# B&R Automation Studio project reAM250plc (part 3)

#### IOModule_X20AT6402.hpp
```cpp
/*++

Copyright (C) 2024 Institute for Machine Tools and Industrial Management
TUM School of Engineering and Design
Technical University of Munich

All rights reserved.

Redistribution and use in source and binary forms, with or without
modification, are permitted provided that the following conditions are met:
	* Redistributions of source code must retain the above copyright
	  notice, this list of conditions and the following disclaimer.
	* Redistributions in binary form must reproduce the above copyright
	  notice, this list of conditions and the following disclaimer in the
	  documentation and/or other materials provided with the distribution.
	* Neither the name of the Technical University of Munich nor the
	  names of its contributors may be used to endorse or promote products
	  derived from this software without specific prior written permission.

THIS SOFTWARE IS PROVIDED BY THE COPYRIGHT HOLDERS AND CONTRIBUTORS "AS IS" AND
ANY EXPRESS OR IMPLIED WARRANTIES, INCLUDING, BUT NOT LIMITED TO, THE IMPLIED
WARRANTIES OF MERCHANTABILITY AND FITNESS FOR A PARTICULAR PURPOSE ARE
DISCLAIMED. IN NO EVENT SHALL TECHNICAL UNIVERSITY OF MUNICH BE LIABLE FOR ANY
DIRECT, INDIRECT, INCIDENTAL, SPECIAL, EXEMPLARY, OR CONSEQUENTIAL DAMAGES
(INCLUDING, BUT NOT LIMITED TO, PROCUREMENT OF SUBSTITUTE GOODS OR SERVICES;
LOSS OF USE, DATA, OR PROFITS; OR BUSINESS INTERRUPTION) HOWEVER CAUSED AND
ON ANY THEORY OF LIABILITY, WHETHER IN CONTRACT, STRICT LIABILITY, OR TORT
(INCLUDING NEGLIGENCE OR OTHERWISE) ARISING IN ANY WAY OUT OF THE USE OF THIS
SOFTWARE, EVEN IF ADVISED OF THE POSSIBILITY OF SUCH DAMAGE.

*/

#ifndef __IOMODULE_X20AT6402_HPP
#define __IOMODULE_X20AT6402_HPP

#include "../Framework/Framework.hpp"

namespace BuRCPP {

	enum class eIOModuleType_X20AT6402 : uint32_t {
		mtUnknown = 0,
		mtVoltage10V = 1,
		mtCurrent20mA = 2,
		mtCurrent24mA = 3
	};

	class CIOModule_X20AT6402 : public CIOModule {
		protected:
		IOMappingX20AT6402_TYP * m_pMapping;
		eIOModuleType_X20AT6402 m_ModuleType;
		int16_t m_nLowerLimit;
		int16_t m_nUpperLimit;

		public:
		CIOModule_X20AT6402 (const std::string & sName, IOMappingX20AT6402_TYP * pMapping);
		virtual ~CIOModule_X20AT6402 ();

		bool isActive () override;
		uint32_t getSerialNumber () override;
		uint16_t getModuleID () override;
		uint16_t getHardwareVariant () override;
		uint16_t getFirmwareVersion () override;

		int16_t getRawValue (uint32_t nChannelNo);
		;
		uint16_t getIOStatus (uint32_t nChannelNo);

		virtual void onRegisterJournal () override;
		virtual void onUpdateJournal () override;

	};

}

#endif //__IOMODULE_X20AT6402_HPP
```

#### IOModule_X20AT6402.cpp
```cpp
/*++

Copyright (C) 2024 Institute for Machine Tools and Industrial Management
TUM School of Engineering and Design
Technical University of Munich

All rights reserved.

Redistribution and use in source and binary forms, with or without
modification, are permitted provided that the following conditions are met:
	* Redistributions of source code must retain the above copyright
	  notice, this list of conditions and the following disclaimer.
	* Redistributions in binary form must reproduce the above copyright
	  notice, this list of conditions and the following disclaimer in the
	  documentation and/or other materials provided with the distribution.
	* Neither the name of the Technical University of Munich nor the
	  names of its contributors may be used to endorse or promote products
	  derived from this software without specific prior written permission.

THIS SOFTWARE IS PROVIDED BY THE COPYRIGHT HOLDERS AND CONTRIBUTORS "AS IS" AND
ANY EXPRESS OR IMPLIED WARRANTIES, INCLUDING, BUT NOT LIMITED TO, THE IMPLIED
WARRANTIES OF MERCHANTABILITY AND FITNESS FOR A PARTICULAR PURPOSE ARE
DISCLAIMED. IN NO EVENT SHALL TECHNICAL UNIVERSITY OF MUNICH BE LIABLE FOR ANY
DIRECT, INDIRECT, INCIDENTAL, SPECIAL, EXEMPLARY, OR CONSEQUENTIAL DAMAGES
(INCLUDING, BUT NOT LIMITED TO, PROCUREMENT OF SUBSTITUTE GOODS OR SERVICES;
LOSS OF USE, DATA, OR PROFITS; OR BUSINESS INTERRUPTION) HOWEVER CAUSED AND
ON ANY THEORY OF LIABILITY, WHETHER IN CONTRACT, STRICT LIABILITY, OR TORT
(INCLUDING NEGLIGENCE OR OTHERWISE) ARISING IN ANY WAY OUT OF THE USE OF THIS
SOFTWARE, EVEN IF ADVISED OF THE POSSIBILITY OF SUCH DAMAGE.

*/

#include "IOModule_X20AT6402.hpp"

// Raw Registers
#define JOURNALVARIABLE_X20AT6402_MODULEOK 1
#define JOURNALVARIABLE_X20AT6402_SERIALNUMBER 2
#define JOURNALVARIABLE_X20AT6402_MODULEID 3
#define JOURNALVARIABLE_X20AT6402_HARDWAREVARIANT 4
#define JOURNALVARIABLE_X20AT6402_FIRMWAREVERSION 5
#define JOURNALVARIABLE_X20AT6402_TEMPERATURE01 6
#define JOURNALVARIABLE_X20AT6402_TEMPERATURE02 7
#define JOURNALVARIABLE_X20AT6402_TEMPERATURE03 8
#define JOURNALVARIABLE_X20AT6402_TEMPERATURE04 9
#define JOURNALVARIABLE_X20AT6402_TEMPERATURE05 10
#define JOURNALVARIABLE_X20AT6402_TEMPERATURE06 11
#define JOURNALVARIABLE_X20AT6402_STATUSINPUT01 12
#define JOURNALVARIABLE_X20AT6402_STATUSINPUT02 13

namespace BuRCPP {

	CIOModule_X20AT6402	::CIOModule_X20AT6402 (const std::string & sName, IOMappingX20AT6402_TYP * pMapping)
		: CIOModule (sName), m_pMapping (pMapping)
	{

	}

	CIOModule_X20AT6402::~CIOModule_X20AT6402 ()
	{
	}

	void CIOModule_X20AT6402::onRegisterJournal ()
	{
		registerBoolValue ("ModuleOk", JOURNALVARIABLE_X20AT6402_MODULEOK);
		registerUInt32Value ("SerialNumber", JOURNALVARIABLE_X20AT6402_SERIALNUMBER);
		registerUInt16Value ("ModuleID", JOURNALVARIABLE_X20AT6402_MODULEID);
		registerUInt16Value ("HardwareVariant", JOURNALVARIABLE_X20AT6402_HARDWAREVARIANT);
		registerUInt16Value ("FirmwareVersion", JOURNALVARIABLE_X20AT6402_FIRMWAREVERSION);
		registerInt16Value ("Temperature01", JOURNALVARIABLE_X20AT6402_TEMPERATURE01);
		registerInt16Value ("Temperature02", JOURNALVARIABLE_X20AT6402_TEMPERATURE02);
		registerInt16Value ("Temperature03", JOURNALVARIABLE_X20AT6402_TEMPERATURE03);
		registerInt16Value ("Temperature04", JOURNALVARIABLE_X20AT6402_TEMPERATURE04);
		registerInt16Value ("Temperature05", JOURNALVARIABLE_X20AT6402_TEMPERATURE05);
		registerInt16Value ("Temperature06", JOURNALVARIABLE_X20AT6402_TEMPERATURE06);
		registerUInt8Value ("StatusInput01", JOURNALVARIABLE_X20AT6402_STATUSINPUT01);
		registerUInt8Value ("StatusInput02", JOURNALVARIABLE_X20AT6402_STATUSINPUT02);
	}

	void CIOModule_X20AT6402::onUpdateJournal ()
	{
		setBoolValue (JOURNALVARIABLE_X20AT6402_MODULEOK, m_pMapping->ModuleOk);
		setIntegerValue (JOURNALVARIABLE_X20AT6402_SERIALNUMBER, m_pMapping->SerialNumber);
		setIntegerValue (JOURNALVARIABLE_X20AT6402_MODULEID, m_pMapping->ModuleID);
		setIntegerValue (JOURNALVARIABLE_X20AT6402_HARDWAREVARIANT, m_pMapping->HardwareVariant);
		setIntegerValue (JOURNALVARIABLE_X20AT6402_FIRMWAREVERSION, m_pMapping->FirmwareVersion);
		setIntegerValue (JOURNALVARIABLE_X20AT6402_TEMPERATURE01, m_pMapping->Temperature01);
		setIntegerValue (JOURNALVARIABLE_X20AT6402_TEMPERATURE02, m_pMapping->Temperature02);
		setIntegerValue (JOURNALVARIABLE_X20AT6402_TEMPERATURE03, m_pMapping->Temperature03);
		setIntegerValue (JOURNALVARIABLE_X20AT6402_TEMPERATURE04, m_pMapping->Temperature04);
		setIntegerValue (JOURNALVARIABLE_X20AT6402_TEMPERATURE05, m_pMapping->Temperature05);
		setIntegerValue (JOURNALVARIABLE_X20AT6402_TEMPERATURE06, m_pMapping->Temperature06);
		setIntegerValue (JOURNALVARIABLE_X20AT6402_STATUSINPUT01, m_pMapping->StatusInput01);
		setIntegerValue (JOURNALVARIABLE_X20AT6402_STATUSINPUT02, m_pMapping->StatusInput02);
	}

	bool CIOModule_X20AT6402::isActive ()
	{
		return m_pMapping->ModuleOk != 0;
	}

	uint32_t CIOModule_X20AT6402::getSerialNumber ()
	{
		return m_pMapping->SerialNumber;
	}

	uint16_t CIOModule_X20AT6402::getModuleID ()
	{
		return m_pMapping->ModuleID;
	}

	uint16_t CIOModule_X20AT6402::getHardwareVariant ()
	{
		return m_pMapping->HardwareVariant;
	}

	uint16_t CIOModule_X20AT6402::getFirmwareVersion ()
	{
		return m_pMapping->FirmwareVersion;
	}

	int16_t CIOModule_X20AT6402::getRawValue (uint32_t nChannelNo)
	{

		switch (nChannelNo) {
			case 1: return m_pMapping->Temperature01;
			case 2: return m_pMapping->Temperature02;
			case 3: return m_pMapping->Temperature03;
			case 4: return m_pMapping->Temperature04;
			case 5: return m_pMapping->Temperature05;
			case 6: return m_pMapping->Temperature06;
			default:
				throw CException (eErrorCode::INVALIDCHANNELNUMBER, "invalid channel number: " + std::to_string (nChannelNo));
		}
	}

	uint16_t CIOModule_X20AT6402::getIOStatus (uint32_t nChannelNo)
	{
		//status IDs: 0 = no error, 1 = lower limit value undershot, 2 = upper limit value exceeded, 3 = wire breakage
		switch (nChannelNo) {
			case 1: return (m_pMapping->StatusInput01 & 0x03);
			case 2: return ((m_pMapping->StatusInput01 >> 2) & 0x03);
			case 3: return ((m_pMapping->StatusInput01 >> 4) & 0x03);
			case 4: return ((m_pMapping->StatusInput01 >> 6) & 0x03);
			case 5: return (m_pMapping->StatusInput02 & 0x03);
			case 6: return ((m_pMapping->StatusInput02 >> 2) & 0x03);
			default:
				throw CException (eErrorCode::INVALIDCHANNELNUMBER, "invalid channel number: " + std::to_string (nChannelNo));
		}
	}

}
```

#### MappMotion_SingleAxis.hpp
```cpp
/*++

Copyright (C) 2024 Institute for Machine Tools and Industrial Management
TUM School of Engineering and Design
Technical University of Munich

All rights reserved.

Redistribution and use in source and binary forms, with or without
modification, are permitted provided that the following conditions are met:
	* Redistributions of source code must retain the above copyright
	  notice, this list of conditions and the following disclaimer.
	* Redistributions in binary form must reproduce the above copyright
	  notice, this list of conditions and the following disclaimer in the
	  documentation and/or other materials provided with the distribution.
	* Neither the name of the Technical University of Munich nor the
	  names of its contributors may be used to endorse or promote products
	  derived from this software without specific prior written permission.

THIS SOFTWARE IS PROVIDED BY THE COPYRIGHT HOLDERS AND CONTRIBUTORS "AS IS" AND
ANY EXPRESS OR IMPLIED WARRANTIES, INCLUDING, BUT NOT LIMITED TO, THE IMPLIED
WARRANTIES OF MERCHANTABILITY AND FITNESS FOR A PARTICULAR PURPOSE ARE
DISCLAIMED. IN NO EVENT SHALL TECHNICAL UNIVERSITY OF MUNICH BE LIABLE FOR ANY
DIRECT, INDIRECT, INCIDENTAL, SPECIAL, EXEMPLARY, OR CONSEQUENTIAL DAMAGES
(INCLUDING, BUT NOT LIMITED TO, PROCUREMENT OF SUBSTITUTE GOODS OR SERVICES;
LOSS OF USE, DATA, OR PROFITS; OR BUSINESS INTERRUPTION) HOWEVER CAUSED AND
ON ANY THEORY OF LIABILITY, WHETHER IN CONTRACT, STRICT LIABILITY, OR TORT
(INCLUDING NEGLIGENCE OR OTHERWISE) ARISING IN ANY WAY OUT OF THE USE OF THIS
SOFTWARE, EVEN IF ADVISED OF THE POSSIBILITY OF SUCH DAMAGE.

*/

#ifndef __MAPPMOTION_SINGLEAXIS_HPP
#define __MAPPMOTION_SINGLEAXIS_HPP

#include "../Framework/Framework.hpp"
#include <memory>

namespace BuRCPP {

	class CMappMotion_SingleAxisImpl;

	enum class eMappMotion_SingleAxisType : int32_t {
		mtLinearAxis = 0,
		mtRotationalAxis = 1,
	};

//	enum class eMappMotion_SingleLinearAxisHomingMode : int32_t {
//		mtDefault = 0,
//		mtRestorePosition = 1,
//	};

	enum class eMappMotion_SingleAxisState : int32_t {
		UNKNOWN = 0,
		STATE_IDLE = 1,
		STATE_SETTINGPOWERON = 2,
		STATE_SETTINGPOWEROFF = 3,
		STATE_REFERENCING = 4,
		STATE_INITABSOLUTEMOVEMENT = 5,
		STATE_INITRELATIVEMOVEMENT = 6,
		STATE_INITVELOCITYMOVEMENT = 7,
		STATE_WAITINGFORMOVEMENT = 8,
		STATE_SETTINGPOWERON_TO_REFERENCE = 9,
		STATE_ERROR = 255,
	};

	class CMappMotion_SingleAxis : public CAxisModule {
		protected:
		McHomingModeEnum m_HomingMode;

		std::shared_ptr<CMappMotion_SingleAxisImpl> m_pImpl;
		eMappMotion_SingleAxisType m_Type;
		eMappMotion_SingleAxisState m_State;

		double m_dSpeedInMMperSecondToSet;
		double m_dAccelerationInMMPerSecondSquaredToSet;
		double m_dTargetPositionInMMToSet;
		double m_dDistanceInMMToSet;

		double m_dSpeedInDegreeperSecondToSet;
		double m_dAccelerationInDegreePerSecondSquaredToSet;
		double m_dTargetPositionInDegreeToSet;
		double m_dDistanceInDegreeToSet;

		public:

		CMappMotion_SingleAxis (const std::string & sName, void * pLink);
		virtual ~CMappMotion_SingleAxis ();

		bool isActive () override;
		bool isIdle ();

		virtual ePLCOpenAxisState getPLCOpenState () override;
		virtual bool isPowered () override;
		virtual bool isReferenced () override;
		virtual bool isMoving () override;
	//	virtual bool isMoveDone () override;

		virtual bool canSetPower () override;
		virtual void setPower (bool bPowerOn) override;

		virtual bool canReference () override;
		virtual void startReference () override;

		virtual void setPowerOnAndStartReference () override;

		void setHomingMode (McHomingModeEnum homingMode);

		virtual bool canMoveAxis ();

		void resetError ();
		void moveAxisReset ();
		bool isError ();
		bool isInPosition ();

		virtual void handleCyclic () override;

		virtual void * getFunctionBlockPtr ();

		virtual void * getParameterBlockPtr ();

		virtual void onRegisterJournal () override;
		virtual void onUpdateJournal () override;

	};

	class CMappMotion_SingleRotationalAxis : public CMappMotion_SingleAxis
	{
		private:

		double m_dMinSpeedInDegreeperSecond;
		double m_dMaxSpeedInDegreeperSecond;

		double m_dMinAccelerationInDegreeperSecond;
		double m_dMaxAccelerationInDegreeperSecond;

		public:

		CMappMotion_SingleRotationalAxis (const std::string & sName, void * pLink);
		virtual ~CMappMotion_SingleRotationalAxis ();

		void moveAxisAbsolute (double targetPositionInDegree, double speedInDegreeperSecond, double accelerationinDegreeSecondsSquared);
		void moveAxisRelative (double targetPositionInDegree, double speedInDegreeperSecond, double accelerationinDegreeSecondsSquared);
		void moveAxisVelocity (double speedInDegreeperSecond, double accelerationinDegreeSecondsSquared);

		double getCurrentPositionInDegree ();
		double getCurrentVelocityInDegreePerSecond ();
	};
	class CMappMotion_SingleLinearAxis : public CMappMotion_SingleAxis
	{
		private:

		double m_dMinSpeedInMMperSecond;
		double m_dMaxSpeedInMMperSecond;

		double m_dMinAccelerationInMMperSecond;
		double m_dMaxAccelerationInMMperSecond;

		public:

		CMappMotion_SingleLinearAxis (const std::string & sName, void * pLink);
		virtual ~CMappMotion_SingleLinearAxis ();

		void moveAxisAbsolute (double targetPositionInMM, double speedInMMperSecond, double accelerationInMMPerSecondSquared);
		void moveAxisRelative (double targetPositionInMM, double speedInMMperSecond, double accelerationInMMPerSecondSquared);
		void moveAxisVelocity (double speedInMMperSecond, double accelerationInMMPerSecondSquared);

		double getCurrentPositionInMM ();
		double getCurrentVelocityInMMPerSecond ();

	};

}

#endif // __MAPPMOTION_SINGLEAXIS_HPP
```

#### MappMotion_SingleAxis.cpp
```cpp
/*++

Copyright (C) 2024 Institute for Machine Tools and Industrial Management
TUM School of Engineering and Design
Technical University of Munich

All rights reserved.

Redistribution and use in source and binary forms, with or without
modification, are permitted provided that the following conditions are met:
	* Redistributions of source code must retain the above copyright
	  notice, this list of conditions and the following disclaimer.
	* Redistributions in binary form must reproduce the above copyright
	  notice, this list of conditions and the following disclaimer in the
	  documentation and/or other materials provided with the distribution.
	* Neither the name of the Technical University of Munich nor the
	  names of its contributors may be used to endorse or promote products
	  derived from this software without specific prior written permission.

THIS SOFTWARE IS PROVIDED BY THE COPYRIGHT HOLDERS AND CONTRIBUTORS "AS IS" AND
ANY EXPRESS OR IMPLIED WARRANTIES, INCLUDING, BUT NOT LIMITED TO, THE IMPLIED
WARRANTIES OF MERCHANTABILITY AND FITNESS FOR A PARTICULAR PURPOSE ARE
DISCLAIMED. IN NO EVENT SHALL TECHNICAL UNIVERSITY OF MUNICH BE LIABLE FOR ANY
DIRECT, INDIRECT, INCIDENTAL, SPECIAL, EXEMPLARY, OR CONSEQUENTIAL DAMAGES
(INCLUDING, BUT NOT LIMITED TO, PROCUREMENT OF SUBSTITUTE GOODS OR SERVICES;
LOSS OF USE, DATA, OR PROFITS; OR BUSINESS INTERRUPTION) HOWEVER CAUSED AND
ON ANY THEORY OF LIABILITY, WHETHER IN CONTRACT, STRICT LIABILITY, OR TORT
(INCLUDING NEGLIGENCE OR OTHERWISE) ARISING IN ANY WAY OUT OF THE USE OF THIS
SOFTWARE, EVEN IF ADVISED OF THE POSSIBILITY OF SUCH DAMAGE.

*/
#include "MappMotion_SingleAxis.hpp"

#include <bur/plctypes.h>

#ifdef _DEFAULT_INCLUDES
#include <AsDefault.h>
#endif

#include <string.h>

#define MAPPMOTION_LINEARAXIS_DEFAULTMINSPEED_IN_MMPERSECOND 0.001f
#define MAPPMOTION_LINEARAXIS_DEFAULTMAXSPEED_IN_MMPERSECOND 1000000.0f
#define MAPPMOTION_LINEARAXIS_DEFAULTMINACCELERATION_IN_MMPERSECONDSQUARED 0.001f
#define MAPPMOTION_LINEARAXIS_DEFAULTMAXACCELERATION_IN_MMPERSECONDSQUARED 1000000.0f

#define MAPPMOTION_ROTARYAXIS_DEFAULTMINSPEED_IN_DEGREEPERSECOND 0.001f
#define MAPPMOTION_ROTARYAXIS_DEFAULTMAXSPEED_IN_DEGREEPERSECOND 1000000.0f
#define MAPPMOTION_ROTARYAXIS_DEFAULTMINACCELERATION_IN_DEGREEPERSECONDSQUARED 0.001f
#define MAPPMOTION_ROTARYAXIS_DEFAULTMAXACCELERATION_IN_DEGREEPERSECONDSQUARED 1000000.0f

#define JOURNALVARIABLE_AXIS_PLCOPENSTATE 1
#define JOURNALVARIABLE_AXIS_CANSETPOWER 2
#define JOURNALVARIABLE_AXIS_ISPOWERED 3
#define JOURNALVARIABLE_AXIS_ISREFERENCED 4
#define JOURNALVARIABLE_AXIS_ISMOVING 5
#define JOURNALVARIABLE_AXIS_ISINPOSITION 6
#define JOURNALVARIABLE_AXIS_ACTUALPOSITION 7
#define JOURNALVARIABLE_AXIS_ACTUALVELOCITY 8

namespace BuRCPP {

	class CMappMotion_SingleAxisImpl {
		private:
		MpAxisBasicParType m_Parameters;
		MpAxisBasic_typ m_FunctionBlock;
		public:

		CMappMotion_SingleAxisImpl (McAxisType * pLink)
		{
			memset ((void*) &m_Parameters, 0, sizeof (MpAxisBasicParType));
			memset ((void*) &m_FunctionBlock, 0, sizeof (MpAxisBasic_typ));

			m_FunctionBlock.MpLink = pLink;
			m_FunctionBlock.Parameters = &m_Parameters;
			m_FunctionBlock.Enable = true;
		}

		virtual ~CMappMotion_SingleAxisImpl ()
		{
			memset ((void*) &m_Parameters, 0, sizeof (MpAxisBasicParType));
			memset ((void*) &m_FunctionBlock, 0, sizeof (MpAxisBasic_typ));
		}

		int32_t getPLCOpenState () const
		{
			return m_FunctionBlock.Info.PLCopenState;
		}

		bool isError () const
		{
			return m_FunctionBlock.Error;
		}

		bool canSetPower () const
		{
			return m_FunctionBlock.Info.ReadyToPowerOn;
		}

		bool isPowered () const
		{
			return m_FunctionBlock.PowerOn;
		}

		bool isReferenced () const
		{
			return m_FunctionBlock.IsHomed;
		}

		bool isMoving () const
		{
			return m_FunctionBlock.MoveActive;
		}

		bool isInPosition () const
		{
			return m_FunctionBlock.InPosition;
		}

		float getCurrentPosition () const
		{
			return m_FunctionBlock.Position;
		}

		float getCurrentVelocity () const
		{
			return m_FunctionBlock.Velocity;
		}

		void setErrorResetFlag (bool bErrorResetFlag)
		{
			m_FunctionBlock.ErrorReset = bErrorResetFlag;
		}

		void setPowerFlag (bool bPowerFlag)
		{
			m_FunctionBlock.Power = bPowerFlag;
		}

		void setHomeFlag (bool bHomeFlag)
		{
			m_FunctionBlock.Home = bHomeFlag;
		}

		void setVelocityParameter (float fVelocity)
		{
			m_Parameters.Velocity = fVelocity;
		}

		void setAccelerationDecelerationParameter (float fAccelerationDeceleration)
		{
			m_Parameters.Acceleration = fAccelerationDeceleration;
			m_Parameters.Deceleration = fAccelerationDeceleration;
		}

		void setAbsoluteMovementTarget (float fTargetPosition)
		{
			m_Parameters.Position = fTargetPosition;
		}

		void setAbsoluteMovementFlag (bool bMovementFlag)
		{
			m_FunctionBlock.MoveAbsolute = bMovementFlag;
		}

		void setRelativeMovementDistance (float fRelativeDistance)
		{
			m_Parameters.Distance = fRelativeDistance;
		}

		void setRelativeMovementFlag (bool bMovementFlag)
		{
			m_FunctionBlock.MoveAdditive = bMovementFlag;
		}

		void setVelocityMovementFlag (bool bMovementFlag)
		{
			m_FunctionBlock.MoveVelocity = bMovementFlag;
		}

		void setHomingMode (McHomingModeEnum homingMode)
		{
			m_Parameters.Homing.Mode = homingMode;
		}

		void handleCyclic ()
		{
			MpAxisBasic(&m_FunctionBlock);
		}

		void * getFunctionBlockPtr ()
		{
			return &m_FunctionBlock;
		}

		void * getParameterBlockPtr ()
		{
			return &m_Parameters;
		}

	};

	CMappMotion_SingleAxis::CMappMotion_SingleAxis (const std::string & sName, void * pLink)
		: CAxisModule (sName),
		m_State (eMappMotion_SingleAxisState::STATE_IDLE),
		m_dSpeedInMMperSecondToSet (0.0),
		m_dAccelerationInMMPerSecondSquaredToSet (0.0),
		m_dTargetPositionInMMToSet (0.0),
		m_dDistanceInMMToSet (0.0)
	{
		m_HomingMode = mcHOMING_DEFAULT;

		if (pLink == nullptr)
			throw CException (eErrorCode::INVALIDAXISLINK, "invalid axis link: " + sName);
/*	if (pFunctionBlock == nullptr)
		throw CException (eErrorCode::INVALIDFUNCTIONBLOCK, "invalid axis function block: " + sName);
	if (pParameterBlock == nullptr)
		throw CException (eErrorCode::INVALIDPARAMETERBLOCK, "invalid axis parameter block: " + sName);*/

		m_pImpl.reset ( new CMappMotion_SingleAxisImpl ((McAxisType*) pLink) );

		// TODO: Read out speed and acceleration limits...
	}

	CMappMotion_SingleAxis::~CMappMotion_SingleAxis ()
	{
	}

	void * CMappMotion_SingleAxis::getFunctionBlockPtr ()
	{
		return m_pImpl->getFunctionBlockPtr ();
	}

	void * CMappMotion_SingleAxis::getParameterBlockPtr ()
	{
		return m_pImpl->getParameterBlockPtr ();
	}

	bool CMappMotion_SingleAxis::isActive ()
	{
		return true;
	}

	ePLCOpenAxisState CMappMotion_SingleAxis::getPLCOpenState ()
	{
		return (ePLCOpenAxisState) m_pImpl->getPLCOpenState ();

	}

	bool CMappMotion_SingleAxis::isIdle ()
	{
		return (m_State == eMappMotion_SingleAxisState::STATE_IDLE);
	}

	bool CMappMotion_SingleAxis::isPowered ()
	{
		return m_pImpl->isPowered ();
	}

	bool CMappMotion_SingleAxis::isReferenced ()
	{
		return m_pImpl->isReferenced ();
	}

	bool CMappMotion_SingleAxis::isMoving ()
	{
		return m_pImpl->isMoving ();
	}

	bool CMappMotion_SingleAxis::isInPosition ()
	{
		return m_pImpl->isInPosition ();
	}

	bool CMappMotion_SingleAxis::canSetPower ()
	{
		return m_pImpl->canSetPower ();
	}

	bool CMappMotion_SingleAxis::isError ()
	{
		return m_pImpl->isError ();
	}

	void CMappMotion_SingleAxis::setPower (bool bPowerOn)
	{
		if (bPowerOn) {
			if (canSetPower ()) {
				m_pImpl->setPowerFlag (true);
				m_State = eMappMotion_SingleAxisState::STATE_SETTINGPOWERON;
			} else {
				throw CException (eErrorCode::COULDNOTPOWERAXIS, "could not power axis: " + m_sName);
			}

		}
		else {
			if (isIdle ()) {
				m_pImpl->setPowerFlag (false);
				m_State = eMappMotion_SingleAxisState::STATE_SETTINGPOWEROFF;

			} else {
				throw CException (eErrorCode::COULDNOTPOWERAXIS, "could not gracefully unpower axis: " + m_sName);
			}
		}

	}

	bool CMappMotion_SingleAxis::canReference ()
	{
		if (isIdle () && isPowered () && (m_pImpl->getPLCOpenState () == mcAXIS_STANDSTILL)) {
			return true;
		} else {
			return false;
		}
	}

	void CMappMotion_SingleAxis::startReference ()
	{
		if (canReference ()) {

			if (DiagCpuIsSimulated()) {
				m_HomingMode = mcHOMING_DIRECT;
				m_pImpl->setHomingMode(m_HomingMode);

			}
			else
			{
				m_pImpl->setHomingMode(m_HomingMode);
			}

			m_pImpl->setHomeFlag (true);
			m_State = eMappMotion_SingleAxisState::STATE_REFERENCING;

		} else {

			throw CException (eErrorCode::COULDNOTREFERENCEAXIS, "could not reference axis: " + m_sName);

		}
	}

	void CMappMotion_SingleAxis::setHomingMode (McHomingModeEnum homingMode)
	{
		m_HomingMode = homingMode;
		m_pImpl->setHomingMode(m_HomingMode);
	}

	void CMappMotion_SingleAxis::setPowerOnAndStartReference ()
	{
		if (canSetPower ()) {
			m_pImpl->setPowerFlag (true);
			m_State = eMappMotion_SingleAxisState::STATE_SETTINGPOWERON_TO_REFERENCE;
		} else {
			throw CException (eErrorCode::COULDNOTPOWERAXIS, "could not power axis: " + m_sName);
		}
	}

	bool CMappMotion_SingleAxis::canMoveAxis ()
	{
		if (isIdle () && isPowered () && isReferenced() && (m_pImpl->getPLCOpenState () == mcAXIS_STANDSTILL)) {
			return true;
		} else {
			return false;
		}
	}

	void CMappMotion_SingleAxis::resetError ()
	{
		if (m_pImpl->isError ()) {
			m_pImpl->setPowerFlag(false);
			m_pImpl->setErrorResetFlag (true);
		}
		else{
			m_pImpl->setErrorResetFlag (false);
			m_pImpl->setPowerFlag(true);
			m_State = eMappMotion_SingleAxisState::STATE_SETTINGPOWERON;
		}

	}

	void CMappMotion_SingleAxis::moveAxisReset ()
	{
		m_pImpl->setVelocityMovementFlag(false);
		m_pImpl->setAbsoluteMovementFlag(false);
		m_pImpl->setRelativeMovementFlag(false);
	}

	void CMappMotion_SingleAxis::onRegisterJournal ()
	{
		registerUInt16Value ("PlcOpenState", JOURNALVARIABLE_AXIS_PLCOPENSTATE);
		registerBoolValue ("CanSetPower", JOURNALVARIABLE_AXIS_CANSETPOWER);
		registerBoolValue ("IsPowered", JOURNALVARIABLE_AXIS_ISPOWERED);
		registerBoolValue ("IsReferenced", JOURNALVARIABLE_AXIS_ISREFERENCED);
		registerBoolValue ("IsMoving", JOURNALVARIABLE_AXIS_ISMOVING);
		registerBoolValue ("IsInPosition", JOURNALVARIABLE_AXIS_ISINPOSITION);
		registerDoubleValue ("ActualPosition", JOURNALVARIABLE_AXIS_ACTUALPOSITION, -1000000, 1000000, 1);
		registerDoubleValue ("ActualVelocity", JOURNALVARIABLE_AXIS_ACTUALVELOCITY, -1000000, 1000000, 1);

	}

void CMappMotion_SingleAxis::onUpdateJournal ()
	{
		setIntegerValue (JOURNALVARIABLE_AXIS_PLCOPENSTATE, m_pImpl->getPLCOpenState());
		setBoolValue (JOURNALVARIABLE_AXIS_CANSETPOWER, canSetPower());
		setBoolValue (JOURNALVARIABLE_AXIS_ISPOWERED, isPowered());
		setBoolValue (JOURNALVARIABLE_AXIS_ISREFERENCED, isReferenced());
		setBoolValue (JOURNALVARIABLE_AXIS_ISMOVING, isMoving());
		setBoolValue (JOURNALVARIABLE_AXIS_ISINPOSITION,  isInPosition());
		setDoubleValue (JOURNALVARIABLE_AXIS_ACTUALPOSITION, m_pImpl->getCurrentPosition());
		setDoubleValue (JOURNALVARIABLE_AXIS_ACTUALVELOCITY, m_pImpl->getCurrentVelocity());

	}

CMappMotion_SingleLinearAxis::CMappMotion_SingleLinearAxis (const std::string & sName, void * pLink)
	: CMappMotion_SingleAxis (sName, pLink),
	m_dMinSpeedInMMperSecond (MAPPMOTION_LINEARAXIS_DEFAULTMINSPEED_IN_MMPERSECOND),
	m_dMaxSpeedInMMperSecond (MAPPMOTION_LINEARAXIS_DEFAULTMAXSPEED_IN_MMPERSECOND),
	m_dMinAccelerationInMMperSecond (MAPPMOTION_LINEARAXIS_DEFAULTMINACCELERATION_IN_MMPERSECONDSQUARED),
	m_dMaxAccelerationInMMperSecond (MAPPMOTION_LINEARAXIS_DEFAULTMAXACCELERATION_IN_MMPERSECONDSQUARED)
{
		m_Type = eMappMotion_SingleAxisType::mtLinearAxis;
}

CMappMotion_SingleLinearAxis::~CMappMotion_SingleLinearAxis ()
{
}

void CMappMotion_SingleLinearAxis::moveAxisAbsolute (double targetPositionInMM, double speedInMMperSecond, double accelerationInMMPerSecondSquared)
{
	if ((speedInMMperSecond < m_dMinSpeedInMMperSecond) || (speedInMMperSecond > m_dMaxSpeedInMMperSecond))
		throw CException (eErrorCode::INVALIDSPEEDVALUE, "invalid speed value for axis: " + m_sName);
	if ((accelerationInMMPerSecondSquared < m_dMinAccelerationInMMperSecond) || (accelerationInMMPerSecondSquared > m_dMaxAccelerationInMMperSecond))
		throw CException (eErrorCode::INVALIDACCELERATIONVALUE, "invalid acceleration value for axis: " + m_sName);

	if (m_State != eMappMotion_SingleAxisState::STATE_IDLE)
		throw CException (eErrorCode::COULDNOTMOVEAXIS, "axis is not in idle mode: " + m_sName);
	if (!canMoveAxis ())
		throw CException (eErrorCode::COULDNOTMOVEAXIS, "could not move axis: " + m_sName);

	m_dTargetPositionInMMToSet = targetPositionInMM;
	m_dSpeedInMMperSecondToSet = speedInMMperSecond;
	m_dAccelerationInMMPerSecondSquaredToSet = accelerationInMMPerSecondSquared;

	m_State = eMappMotion_SingleAxisState::STATE_INITABSOLUTEMOVEMENT;

}

void CMappMotion_SingleLinearAxis::moveAxisRelative (double distanceInMM, double speedInMMperSecond, double accelerationInMMPerSecondSquared)
{
	if ((speedInMMperSecond < m_dMinSpeedInMMperSecond) || (speedInMMperSecond > m_dMaxSpeedInMMperSecond))
		throw CException (eErrorCode::INVALIDSPEEDVALUE, "invalid speed value for axis: " + m_sName);
	if ((accelerationInMMPerSecondSquared < m_dMinAccelerationInMMperSecond) || (accelerationInMMPerSecondSquared > m_dMaxAccelerationInMMperSecond))
		throw CException (eErrorCode::INVALIDACCELERATIONVALUE, "invalid acceleration value for axis: " + m_sName);

	if (m_State != eMappMotion_SingleAxisState::STATE_IDLE)
		throw CException (eErrorCode::COULDNOTMOVEAXIS, "axis is not in idle mode: " + m_sName);
	if (!canMoveAxis ())
		throw CException (eErrorCode::COULDNOTMOVEAXIS, "could not move axis: " + m_sName);

	m_dDistanceInMMToSet = distanceInMM;
	m_dSpeedInMMperSecondToSet = speedInMMperSecond;
	m_dAccelerationInMMPerSecondSquaredToSet = accelerationInMMPerSecondSquared;

	m_State = eMappMotion_SingleAxisState::STATE_INITRELATIVEMOVEMENT;
}

void CMappMotion_SingleLinearAxis::moveAxisVelocity (double speedInMMperSecond, double accelerationInMMPerSecondSquared)
{
	if ((speedInMMperSecond < m_dMinSpeedInMMperSecond) || (speedInMMperSecond > m_dMaxSpeedInMMperSecond))
		throw CException (eErrorCode::INVALIDSPEEDVALUE, "invalid speed value for axis: " + m_sName);
	if ((accelerationInMMPerSecondSquared < m_dMinAccelerationInMMperSecond) || (accelerationInMMPerSecondSquared > m_dMaxAccelerationInMMperSecond))
		throw CException (eErrorCode::INVALIDACCELERATIONVALUE, "invalid acceleration value for axis: " + m_sName);

	if (m_State != eMappMotion_SingleAxisState::STATE_IDLE)
		throw CException (eErrorCode::COULDNOTMOVEAXIS, "axis is not in idle mode: " + m_sName);
	if (!canMoveAxis ())
		throw CException (eErrorCode::COULDNOTMOVEAXIS, "could not move axis: " + m_sName);

	m_dSpeedInMMperSecondToSet = speedInMMperSecond;
	m_dAccelerationInMMPerSecondSquaredToSet = accelerationInMMPerSecondSquared;

	m_State = eMappMotion_SingleAxisState::STATE_INITVELOCITYMOVEMENT;
}

double CMappMotion_SingleLinearAxis::getCurrentPositionInMM ()
{
	return (double) m_pImpl->getCurrentPosition ();
}

double CMappMotion_SingleLinearAxis::getCurrentVelocityInMMPerSecond ()
{
	return (double) m_pImpl->getCurrentVelocity ();
}

CMappMotion_SingleRotationalAxis::CMappMotion_SingleRotationalAxis (const std::string & sName, void * pLink)
	: CMappMotion_SingleAxis (sName, pLink),
	m_dMinSpeedInDegreeperSecond (MAPPMOTION_ROTARYAXIS_DEFAULTMINSPEED_IN_DEGREEPERSECOND),
	m_dMaxSpeedInDegreeperSecond (MAPPMOTION_ROTARYAXIS_DEFAULTMAXSPEED_IN_DEGREEPERSECOND),
	m_dMinAccelerationInDegreeperSecond (MAPPMOTION_ROTARYAXIS_DEFAULTMINACCELERATION_IN_DEGREEPERSECONDSQUARED),
	m_dMaxAccelerationInDegreeperSecond (MAPPMOTION_ROTARYAXIS_DEFAULTMAXACCELERATION_IN_DEGREEPERSECONDSQUARED)
{
		m_Type = eMappMotion_SingleAxisType::mtRotationalAxis;
}

CMappMotion_SingleRotationalAxis::~CMappMotion_SingleRotationalAxis ()
{
}

void CMappMotion_SingleRotationalAxis::moveAxisAbsolute (double targetPositionInDegree, double speedInDegreeperSecond, double accelerationinDegreeSecondsSquared)
{

	if ((speedInDegreeperSecond < m_dMinSpeedInDegreeperSecond) || (speedInDegreeperSecond > m_dMaxSpeedInDegreeperSecond))
		throw CException (eErrorCode::INVALIDSPEEDVALUE, "invalid speed value for axis: " + m_sName);
	if ((accelerationinDegreeSecondsSquared < m_dMinAccelerationInDegreeperSecond) || (accelerationinDegreeSecondsSquared > m_dMaxAccelerationInDegreeperSecond))
		throw CException (eErrorCode::INVALIDACCELERATIONVALUE, "invalid acceleration value for axis: " + m_sName);

	if (m_State != eMappMotion_SingleAxisState::STATE_IDLE)
		throw CException (eErrorCode::COULDNOTMOVEAXIS, "axis is not in idle mode: " + m_sName);
	if (!canMoveAxis ())
		throw CException (eErrorCode::COULDNOTMOVEAXIS, "could not move axis: " + m_sName);

	m_dTargetPositionInDegreeToSet = targetPositionInDegree;
	m_dSpeedInDegreeperSecondToSet = speedInDegreeperSecond;
	m_dAccelerationInDegreePerSecondSquaredToSet = accelerationinDegreeSecondsSquared;

	m_State = eMappMotion_SingleAxisState::STATE_INITABSOLUTEMOVEMENT;

}

void CMappMotion_SingleRotationalAxis::moveAxisRelative (double distanceInDegree, double speedInDegreeperSecond, double accelerationInDegreePerDegreeSecond)
{
	if ((speedInDegreeperSecond < m_dMinSpeedInDegreeperSecond) || (speedInDegreeperSecond > m_dMaxSpeedInDegreeperSecond))
		throw CException (eErrorCode::INVALIDSPEEDVALUE, "invalid speed value for axis: " + m_sName);
	if ((accelerationInDegreePerDegreeSecond < m_dMinAccelerationInDegreeperSecond) || (accelerationInDegreePerDegreeSecond > m_dMaxAccelerationInDegreeperSecond))
		throw CException (eErrorCode::INVALIDACCELERATIONVALUE, "invalid acceleration value for axis: " + m_sName);

	if (m_State != eMappMotion_SingleAxisState::STATE_IDLE)
		throw CException (eErrorCode::COULDNOTMOVEAXIS, "axis is not in idle mode: " + m_sName);
	if (!canMoveAxis ())
		throw CException (eErrorCode::COULDNOTMOVEAXIS, "could not move axis: " + m_sName);

	m_dDistanceInDegreeToSet = distanceInDegree;
	m_dSpeedInDegreeperSecondToSet = speedInDegreeperSecond;
	m_dAccelerationInDegreePerSecondSquaredToSet = accelerationInDegreePerDegreeSecond;

	m_State = eMappMotion_SingleAxisState::STATE_INITRELATIVEMOVEMENT;
}

void CMappMotion_SingleRotationalAxis::moveAxisVelocity (double speedInDegreeperSecond, double accelerationInDegreePerSecondSquared)
{
	if ((speedInDegreeperSecond < m_dMinSpeedInDegreeperSecond) || (speedInDegreeperSecond > m_dMaxSpeedInDegreeperSecond))
		throw CException (eErrorCode::INVALIDSPEEDVALUE, "invalid speed value for axis: " + m_sName);
	if ((accelerationInDegreePerSecondSquared < m_dMinAccelerationInDegreeperSecond) || (accelerationInDegreePerSecondSquared > m_dMaxAccelerationInDegreeperSecond))
		throw CException (eErrorCode::INVALIDACCELERATIONVALUE, "invalid acceleration value for axis: " + m_sName);

	if (m_State != eMappMotion_SingleAxisState::STATE_IDLE)
		throw CException (eErrorCode::COULDNOTMOVEAXIS, "axis is not in idle mode: " + m_sName);
	if (!canMoveAxis ())
		throw CException (eErrorCode::COULDNOTMOVEAXIS, "could not move axis: " + m_sName);

	m_dSpeedInDegreeperSecondToSet = speedInDegreeperSecond;
	m_dAccelerationInDegreePerSecondSquaredToSet = accelerationInDegreePerSecondSquared;

	m_State = eMappMotion_SingleAxisState::STATE_INITVELOCITYMOVEMENT;
}

double CMappMotion_SingleRotationalAxis::getCurrentPositionInDegree ()
{
	return (double) m_pImpl->getCurrentPosition ();
}

double CMappMotion_SingleRotationalAxis::getCurrentVelocityInDegreePerSecond ()
{
	return (double) m_pImpl->getCurrentVelocity ();
}

void CMappMotion_SingleAxis::handleCyclic ()
{

	m_pImpl->handleCyclic ();

	switch (m_State) {
		case eMappMotion_SingleAxisState::STATE_SETTINGPOWERON:

			if (m_pImpl->isPowered ())
				m_State = eMappMotion_SingleAxisState::STATE_IDLE;

			if (m_pImpl->isError ())
				m_State = eMappMotion_SingleAxisState::STATE_ERROR;

			break;

		case eMappMotion_SingleAxisState::STATE_SETTINGPOWERON_TO_REFERENCE:
			if (m_pImpl->isPowered ()) {
				if ((m_pImpl->getPLCOpenState () == mcAXIS_STANDSTILL)) {
						if (DiagCpuIsSimulated()) {
							m_HomingMode = mcHOMING_DIRECT;
							m_pImpl->setHomingMode(m_HomingMode);

						}
						else
						{
							m_pImpl->setHomingMode(m_HomingMode);
						}
						m_pImpl->setHomingMode(m_HomingMode);
						m_pImpl->setHomeFlag (true);
					m_State = eMappMotion_SingleAxisState::STATE_REFERENCING;
				} else {
					m_State = eMappMotion_SingleAxisState::STATE_ERROR;
				}
			}
			if (m_pImpl->isError ())
				m_State = eMappMotion_SingleAxisState::STATE_ERROR;
			break;

		case eMappMotion_SingleAxisState::STATE_SETTINGPOWEROFF:
			if (!m_pImpl->isPowered ())
				m_State = eMappMotion_SingleAxisState::STATE_IDLE;
			if (m_pImpl->isError ())
				m_State = eMappMotion_SingleAxisState::STATE_ERROR;

			break;

		case eMappMotion_SingleAxisState::STATE_REFERENCING:
			if (m_pImpl->isReferenced ()) {
				m_pImpl->setHomeFlag (false);
				m_State = eMappMotion_SingleAxisState::STATE_IDLE;
			}
			if (m_pImpl->isError ()) {
				m_pImpl->setHomeFlag (false);
				m_State = eMappMotion_SingleAxisState::STATE_ERROR;
			}

			break;

		case eMappMotion_SingleAxisState::STATE_INITABSOLUTEMOVEMENT:
			if (m_pImpl->isError ()) {
				m_State = eMappMotion_SingleAxisState::STATE_ERROR;
			} else {
					if(m_Type == eMappMotion_SingleAxisType::mtLinearAxis)
					{
						m_pImpl->setVelocityParameter(m_dSpeedInMMperSecondToSet);
						m_pImpl->setAccelerationDecelerationParameter(m_dAccelerationInMMPerSecondSquaredToSet);
						m_pImpl->setAbsoluteMovementTarget (m_dTargetPositionInMMToSet);
					}
					else if (m_Type == eMappMotion_SingleAxisType::mtRotationalAxis)
					{
						m_pImpl->setVelocityParameter(m_dSpeedInDegreeperSecondToSet);
						m_pImpl->setAccelerationDecelerationParameter(m_dAccelerationInDegreePerSecondSquaredToSet);
						m_pImpl->setAbsoluteMovementTarget (m_dTargetPositionInDegreeToSet);
					}
					m_pImpl->setAbsoluteMovementFlag (true);
					m_State = eMappMotion_SingleAxisState::STATE_WAITINGFORMOVEMENT;
			}

			break;

		case eMappMotion_SingleAxisState::STATE_INITRELATIVEMOVEMENT:
			if (m_pImpl->isError ()) {
				m_State = eMappMotion_SingleAxisState::STATE_ERROR;
			} else {
					if(m_Type == eMappMotion_SingleAxisType::mtLinearAxis)
					{
						m_pImpl->setVelocityParameter(m_dSpeedInMMperSecondToSet);
						m_pImpl->setAccelerationDecelerationParameter(m_dAccelerationInMMPerSecondSquaredToSet);
						m_pImpl->setRelativeMovementDistance (m_dDistanceInMMToSet);
					}
					else if (m_Type == eMappMotion_SingleAxisType::mtRotationalAxis)
					{
						m_pImpl->setVelocityParameter(m_dSpeedInDegreeperSecondToSet);
						m_pImpl->setAccelerationDecelerationParameter(m_dAccelerationInDegreePerSecondSquaredToSet);
						m_pImpl->setRelativeMovementDistance (m_dDistanceInDegreeToSet);
					}
					m_pImpl->setRelativeMovementFlag (true);
					m_State = eMappMotion_SingleAxisState::STATE_WAITINGFORMOVEMENT;
			}

			break;

		case eMappMotion_SingleAxisState::STATE_INITVELOCITYMOVEMENT:
			if (m_pImpl->isError ()) {
				m_State = eMappMotion_SingleAxisState::STATE_ERROR;
			} else {
					if(m_Type == eMappMotion_SingleAxisType::mtLinearAxis)
					{
						m_pImpl->setVelocityParameter(m_dSpeedInMMperSecondToSet);
						m_pImpl->setAccelerationDecelerationParameter(m_dAccelerationInMMPerSecondSquaredToSet);
					}
					else if (m_Type == eMappMotion_SingleAxisType::mtRotationalAxis)
					{
						m_pImpl->setVelocityParameter(m_dSpeedInDegreeperSecondToSet);
						m_pImpl->setAccelerationDecelerationParameter(m_dAccelerationInDegreePerSecondSquaredToSet);
					}
					m_pImpl->setVelocityMovementFlag (true);
					m_State = eMappMotion_SingleAxisState::STATE_WAITINGFORMOVEMENT;
			}

			break;

		case eMappMotion_SingleAxisState::STATE_WAITINGFORMOVEMENT:
			if (m_pImpl->isInPosition ()) {
				m_pImpl->setRelativeMovementFlag (false);
				m_pImpl->setAbsoluteMovementFlag (false);
				m_pImpl->setVelocityMovementFlag (false);
				m_State = eMappMotion_SingleAxisState::STATE_IDLE;
			}
			if (m_pImpl->isError ()) {
				m_pImpl->setRelativeMovementFlag (false);
				m_pImpl->setAbsoluteMovementFlag (false);
				m_pImpl->setVelocityMovementFlag (false);
				m_State = eMappMotion_SingleAxisState::STATE_ERROR;
			}

			break;
	}

}

}
```

#### Framework.hpp
```cpp
/*++

Copyright (C) 2024 Institute for Machine Tools and Industrial Management
TUM School of Engineering and Design
Technical University of Munich

All rights reserved.

Redistribution and use in source and binary forms, with or without
modification, are permitted provided that the following conditions are met:
	* Redistributions of source code must retain the above copyright
	  notice, this list of conditions and the following disclaimer.
	* Redistributions in binary form must reproduce the above copyright
	  notice, this list of conditions and the following disclaimer in the
	  documentation and/or other materials provided with the distribution.
	* Neither the name of the Technical University of Munich nor the
	  names of its contributors may be used to endorse or promote products
	  derived from this software without specific prior written permission.

THIS SOFTWARE IS PROVIDED BY THE COPYRIGHT HOLDERS AND CONTRIBUTORS "AS IS" AND
ANY EXPRESS OR IMPLIED WARRANTIES, INCLUDING, BUT NOT LIMITED TO, THE IMPLIED
WARRANTIES OF MERCHANTABILITY AND FITNESS FOR A PARTICULAR PURPOSE ARE
DISCLAIMED. IN NO EVENT SHALL TECHNICAL UNIVERSITY OF MUNICH BE LIABLE FOR ANY
DIRECT, INDIRECT, INCIDENTAL, SPECIAL, EXEMPLARY, OR CONSEQUENTIAL DAMAGES
(INCLUDING, BUT NOT LIMITED TO, PROCUREMENT OF SUBSTITUTE GOODS OR SERVICES;
LOSS OF USE, DATA, OR PROFITS; OR BUSINESS INTERRUPTION) HOWEVER CAUSED AND
ON ANY THEORY OF LIABILITY, WHETHER IN CONTRACT, STRICT LIABILITY, OR TORT
(INCLUDING NEGLIGENCE OR OTHERWISE) ARISING IN ANY WAY OUT OF THE USE OF THIS
SOFTWARE, EVEN IF ADVISED OF THE POSSIBILITY OF SUCH DAMAGE.

*/

#ifndef __FRAMEWORK_HPP
#define __FRAMEWORK_HPP

#include <cstdint>
#include <memory>
#include <map>
#include <vector>

#include <bur/plctypes.h>

#ifdef _DEFAULT_INCLUDES
#include <AsDefault.h>
#endif

#define COMMAND_DEFAULT_BEGINLIST 101
#define COMMAND_DEFAULT_FINISHLIST 102
#define COMMAND_DEFAULT_EXECUTELIST 103
#define COMMAND_DEFAULT_PAUSELIST 104
#define COMMAND_DEFAULT_LISTSTATUS 105
#define COMMAND_DEFAULT_ABORTLIST 106
#define COMMAND_DEFAULT_RESUMELIST 107
#define COMMAND_DEFAULT_DELETELIST 112
#define COMMAND_DEFAULT_CURRENTJOURNALSTATUS 120
#define COMMAND_DEFAULT_CURRENTJOURNALSCHEMA 121
#define COMMAND_DEFAULT_RETRIEVEJOURNALVARIABLE 122
#define COMMAND_DEFAULT_RETRIEVEJOURNALHISTORY 123

namespace BuRCPP {

	class CJournal;

	enum class eErrorCode : int32_t {
		UNKNOWN = 0,
		INVALIDPARAM = 1,
		STATEALREADYEXISTS = 2,
		STATENOTFOUND = 3,
		NEXTSTATEHASNOTBEENSET = 4,
		MODULEALREADYEXISTS = 5,
		NOVOLTAGEMODULE = 6,
		NOCURRENTMODULE = 7,
		INVALIDCHANNELNUMBER = 8,
		MODULENOTFOUND = 9,
		INVALIDMODULETYPE = 10,
		MODULENOTACTIVE = 11,
		INVALIDAXISLINK = 12,
		COULDNOTPOWERAXIS = 13,
		COULDNOTREFERENCEAXIS = 14,
		INVALIDFUNCTIONBLOCK = 15,
		INVALIDPARAMETERBLOCK = 16,
		INVALIDSPEEDVALUE = 17,
		INVALIDACCELERATIONVALUE = 18,
		COULDNOTMOVEAXIS = 19,
		NOTIMPLEMENTED = 20,
		SERVERISALREADYRUNNING = 21,
		SERVERISNOTRUNNING = 22,
		UNKNOWNTCPSERVERSTATE = 23,
		UNKNOWNTCPRECVSTATE = 24,
		UNKNOWNTCPSENDSTATE = 25,
		INVALIDTCPBUFFERSIZE = 26,
		TCPSENDBUFFERSIZEEXCEEDED = 27,
		TCPSENDBUFFERISFULL = 28,
		PACKETHANDLERALREADYREGISTERED = 29,
		INVALIDPAYLOAD = 30,
		INVALIDTCPRESPONSE = 31,
		NOLISTTOWRITETO = 32,
		LISTEXCEEDSMAXIMUMSIZE = 33,
		TOOMANYOPENLISTS = 34,
		NOLISTENTRIESLEFT = 35,
		INTERNALLISTERROR = 36,
		INVALIDPAYLOADOFFSET = 37,
		INVALIDLISTID = 38,
		LISTISNOTINQUEUE = 39,
		NOTWRITINGTOANYLIST = 40,
		NOTINLISTCREATION = 41,
		LISTISEMPTY = 42,
		LISTDOESNOTEXIST = 43,
		LISTISNOTFINISHED = 44,
		INVALIDNAME = 45,
		DUPLICATESIGNALDEFINITION = 46,
		CANNOTREGISTERSIGNAL = 47,
		CANNOTBUILDSIGNALINSTANCES = 48,
		CANNOTREGISTERPARAMETER = 49,
		SIGNALMEMORYALLOCATIONERROR = 50,
		DUPLICATESIGNALPARAMETERNAME = 51,
		CANNOTREGISTERRESULT = 52,
		DUPLICATESIGNALRESULTNAME = 53,
		INVALIDSIGNALQUEUESIZE = 54,
		SIGNALINSTANCESALREADYBUILT = 55,
		SIGNALDATAMISSINGMEMORY = 56,
		SIGNALDATAWRITEOUTOFRANGE = 57,
		SIGNALDATAREADOUTOFRANGE = 58,
		VALUEISOUTSIDEOFINTEGER32RANGE = 59,
		VALUEISOUTSIDEOFUNSIGNEDINTEGER32RANGE = 60,
		SIGNALPARAMETERNOTFOUND = 61,
		SIGNALRESULTNOTFOUND = 62,
		COULDNOTREADDOUBLEFROMPARAMETER = 63,
		COULDNOTREADINTEGERFROMPARAMETER = 64,
		COULDNOTWRITEDOUBLETOPARAMETER = 65,
		COULDNOTWRITEINTEGERTOPARAMETER = 66,
		INVALIDPAYLOADADDRESS = 67,
		INVALIDPAYLOADREADOPERATION = 68,
		INVALIDCONTEXTADDRESS = 69,
		INVALIDCONTEXTREADOPERATION = 70,
		INVALIDCONTEXTWRITEOPERATION = 71,
		LISTCONTEXT_PAYLOADSIGNALSLOTCOUNT = 72,
		INVALIDSIGNALSLOTINDEX = 73,
		PAYLOADSIGNALSLOTINDEXALREADYTAKEN = 74,
		SIGNALSLOTISEMPTY = 75,
		PAYLOADSIGNALSLOTALREADYTAKEN = 76,
		SIGNALHANDLERNOTFOUND = 77,
		SIGNALHASNOINSTANCES = 78,
		COULDNOTPREPARESIGNAL = 79,
		SIGNALDEFINITIONNOTFOUND = 80,
		COULDNOTCHECKSIGNAL = 81,
		NOSIGNALTOFINISH = 82,
		FINISHEDSIGNALINWRONGORDER = 83,
		SIGNALISNOTINPREPARATION = 84,
		SIGNALISNOTINPROCESS = 85,
		INVALIDREQUEST = 86,
		JOURNALALREADYREGISTERING = 87,
		JOURNALISNOTREGISTERING = 88,
		JOURNALNOTSET = 89,
		EMPTYJOURNALENTRYNAME = 90,
		INVALIDJOURNALENTRYNAME = 91,
		INVALIDJOURNALENTRYID = 92,
		JOURNALISNOTINITIALIZING = 93,
		DUPLICATEJOURNALGROUPID = 94,
		DUPLICATEJOURNALGROUPNAME = 95,
		JOURNALGROUPIDNOTFOUND = 96,
		EMPTYJOURNALGROUPDNAME = 97,
		INVALIDJOURNALGROUPDNAME = 98,
		INVALIDJOURNALGROUPID = 99,
		JOURNALGROUPNAMENOTFOUND = 100,
		EMPTYJOURNALGROUPNAME = 101,
		INVALIDJOURNALGROUPNAME = 102,
		JOURNALENTRYALREADYREGISTERED = 103,
		EMPTYJOURNALNOTALLOWED = 104,
		JOURNALVALUEOUTSIDEOFRANGE = 105,
		JOURNALENTRYTYPEMISMATCH = 106,
		JOURNALENTRYNOTFOUND = 107,
		INVALIDJOURNALADDRESS = 108,
		INVALIDJOURNALENTRYSIZE = 109,
		JOURNALDATABUFFEROVERRUN = 110,
		UNHANDLEDEXCEPTION = 111,
		VARIABLEGROUPNOTFOUND = 112,
		INVALIDENTRYID = 113,
		JOURNALRINGBUFFERISEMPTY = 114,
		JOURNALRINGBUFFERISFULL = 115,
		INVALIDCHANNELTYPE = 116,
		SIGNALTRIGGERTIMEISINFUTURE = 117,
		INVALIDCHANNELVALUE = 118,

	};

	class CStateHandler;
	class CSignalDefinition;
	class CSignalProcessingInstance;
	class CSignalHandler;
	class CState;
	class CEnvironment;
	class CIOModule;
	class CAxisModule;

	class CException {
		private:
		eErrorCode m_Code;
		std::string m_sMessage;

		public:
		CException (eErrorCode code, const std::string & sMessage);
		eErrorCode getCode () const;
		const char * getMessage () const;

	};

	typedef struct _TcpIncomingPayload {
		uint8_t m_Data[24];
	} TcpIncomingPayload;

	typedef struct _TcpIncomingMessage {
		uint32_t m_nSignature;
		uint32_t m_nClientId;
		uint32_t m_nSequenceId;
		uint32_t m_nCommandId;
		TcpIncomingPayload m_Payload;
		uint32_t m_nChecksum;
	} TcpIncomingMessage;

	typedef struct _TcpOutgoingMessageHeader {
		uint32_t m_nSignature;
		uint32_t m_nClientId;
		uint32_t m_nSequenceId;
		uint32_t m_nStatusCode;
		uint32_t m_nPayloadLength;
		uint32_t m_nPayloadChecksum;
		uint32_t m_nHeaderChecksum;
	} TcpOutgoingMessageHeader;

/*

	class CIOChannel {
		private:

		public:

		bool getValue ();

		void setValue (const bool bValue);

		bool isReadOnly ();

		bool hasError ();

		eIOChannelState getState ();

		...

	};

	class CSignleAxisDriver {
		private:

		public:

		bool getValue ();

		void setValue (const bool bValue);

		bool isReadOnly ();

		bool hasError ();

		eIOChannelState getState ();

		...

	};
	 */

	class CModule {
		protected:
		std::string m_sName;
		std::shared_ptr<CJournal> m_pJournal;
		uint32_t m_nJournalGroupID;
		bool m_bJournalIsRegistering;

		public:
		CModule (const std::string & sName);
		virtual ~CModule ();

		virtual std::string getName ();
		virtual bool isActive () = 0;

		virtual void handleCyclic ();

		void setJournal (std::shared_ptr<CJournal> pJournal, uint32_t nJournalGroupID);

		virtual void onRegisterJournal ();
		virtual void onUpdateJournal ();

		void registerIntegerValue (const std::string & sEntryName,const uint32_t nEntryID, int64_t nMinValue, int64_t nMaxValue);
		void registerBoolValue (const std::string & sEntryName,const uint32_t nEntryID);
		void registerDoubleValue (const std::string & sEntryName,const uint32_t nEntryID, double dMinValue, double dMaxValue, int64_t nQuantizationSteps);

		void registerUInt8Value (const std::string & sEntryName,const uint32_t nEntryID);
		void registerUInt16Value (const std::string & sEntryName,const uint32_t nEntryID);
		void registerUInt32Value (const std::string & sEntryName,const uint32_t nEntryID);
		void registerInt8Value (const std::string & sEntryName,const uint32_t nEntryID);
		void registerInt16Value (const std::string & sEntryName,const uint32_t nEntryID);
		void registerInt32Value (const std::string & sEntryName,const uint32_t nEntryID);

		void setIntegerValue (const uint32_t nEntryID, int64_t nValue);
		void setBoolValue (const uint32_t nEntryID, bool bValue);
		void setDoubleValue (const uint32_t nEntryID, double dValue);

	};

	class CIOModule : public CModule {
		public:
		CIOModule (const std::string & sName);
		virtual ~CIOModule ();

		virtual uint32_t getSerialNumber () = 0;
		virtual uint16_t getModuleID () = 0;
		virtual uint16_t getHardwareVariant () = 0;
		virtual uint16_t getFirmwareVersion () = 0;
	};

	enum class ePLCOpenAxisState : int32_t {
		UNKNOWN = 0,
		AXIS_DISABLED = 1,
		AXIS_STANDSTILL = 2,
		AXIS_HOMING = 2,
		AXIS_STOPPING = 3,
		AXIS_DISCRETE_MOTION = 4,
		AXIS_CONTINUOUS_MOTION = 5,
		AXIS_SYNCHRONIZED_MOTION = 6,
		AXIS_ERRORSTOP = 7,
		AXIS_STARTUP = 8,
		AXIS_INVALID_CONFIGURATION = 9
	};

	class CAxisModule : public CModule {
		public:
		CAxisModule (const std::string & sName);
		virtual ~CAxisModule ();

		virtual ePLCOpenAxisState getPLCOpenState () = 0;

		virtual bool isPowered () = 0;
		virtual bool isReferenced () = 0;
		virtual bool isMoving () = 0;

		virtual bool canSetPower () = 0;
		virtual void setPower (bool bPowerOn) = 0;
		void setPowerOn ();
		void setPowerOff ();

		virtual bool canReference () = 0;
		virtual void startReference () = 0;

		virtual void setPowerOnAndStartReference () = 0;

	};

	class CEnvironment {
		private:

		CStateHandler * m_pStateHandler;
		CState * m_pNextState;

		public:

		CEnvironment (CStateHandler * pStateHandler);

		virtual ~CEnvironment ();

		void setNextState (const std::string & sNextState);

		CState * getNextState ();

		CModule * findModule (const std::string & sName, bool bFailIfNotExist);

		CSignalProcessingInstance * checkSignal (const std::string & sName);

		CSignalProcessingInstance * findSignal (uint32_t nSignalID);

		void setIntegerValue (const uint32_t nEntryID, int64_t nValue);
		void setBoolValue (const uint32_t nEntryID, bool bValue);
		void setDoubleValue (const uint32_t nEntryID, double dValue);

		bool getBoolValue (const uint32_t nEntryID);
		double getDoubleValue (const uint32_t nEntryID);
		int64_t getInt64Value (const uint32_t nEntryID);
		int32_t getInt32Value (const uint32_t nEntryID);
		int16_t getInt16Value (const uint32_t nEntryID);
		int8_t getInt8Value (const uint32_t nEntryID);
		uint64_t getUint64Value (const uint32_t nEntryID);
		uint32_t getUint32Value (const uint32_t nEntryID);
		uint16_t getUint16Value (const uint32_t nEntryID);
		uint8_t getUint8Value (const uint32_t nEntryID);

	};

	class CState {

		private:

		public:

		CState ();

		virtual ~CState ();

		virtual std::string getName () = 0;

		virtual void Execute (CEnvironment * pEnvironment) = 0;

	};

	class CModuleHandler {
		private:
			std::map<std::string, std::shared_ptr<CModule>> m_Modules;
			std::shared_ptr<CJournal> m_pJournal;
		public:
			CModuleHandler (std::shared_ptr<CJournal> pJournal);

			virtual ~CModuleHandler ();

			void registerModule (std::shared_ptr<CModule> pModule, uint32_t nJournalGroupID);

			void handleModules ();

			CModule * findModule (const std::string & sName);

	};

	class CStateHandler {
		private:

		std::map<std::string, std::shared_ptr<CState>> m_States;
		std::shared_ptr<CModuleHandler> m_pModuleHandler;

		CState * m_pCurrentState;
		char * m_pStateNameDebug;
		uint32_t m_nStateNameDebugLength;

		std::shared_ptr<CSignalHandler> m_pSignalHandler;
		std::shared_ptr<CJournal> m_pJournal;

		uint32_t m_nJournalGroupID;
		std::string m_sName;

		protected:

		void addState (std::shared_ptr<CState> pState);

		void registerIntegerValue (const std::string & sEntryName,const uint32_t nEntryID, int64_t nMinValue, int64_t nMaxValue);
		void registerBoolValue (const std::string & sEntryName,const uint32_t nEntryID);
		void registerDoubleValue (const std::string & sEntryName,const uint32_t nEntryID, double dMinValue, double dMaxValue, int64_t nQuantizationSteps);

		public:

		CStateHandler (std::shared_ptr<CJournal> pJournal, const std::string & sName, std::shared_ptr<CModuleHandler> pModuleHandler, uint32_t nJournalGroupID);

		virtual ~CStateHandler();

		CState * findState (const std::string & sName);

		CModule * findModule (const std::string & sName);

		CState * getCurrentState ();

		void setCurrentState (CState * pState);

		std::string getName ();

		std::shared_ptr<CSignalDefinition> registerSignal (const std::string & sName, const uint32_t nQueueSize, const uint32_t nLifetimeInMilliseconds);

		void setDebugVariables (char * pStateNameDebug, uint32_t nStateNameDebugLength);
		void writeDebugInformation ();

		virtual void onRegister ();

		CSignalHandler* getSignalHandler ();

		void releaseExpiredSignals ();

		void setIntegerValue (const uint32_t nEntryID, int64_t nValue);
		void setBoolValue (const uint32_t nEntryID, bool bValue);
		void setDoubleValue (const uint32_t nEntryID, double dValue);

		bool getBoolValue (const uint32_t nEntryID);
		double getDoubleValue (const uint32_t nEntryID);
		int64_t getInt64Value (const uint32_t nEntryID);
		int32_t getInt32Value (const uint32_t nEntryID);
		int16_t getInt16Value (const uint32_t nEntryID);
		int8_t getInt8Value (const uint32_t nEntryID);
		uint64_t getUint64Value (const uint32_t nEntryID);
		uint32_t getUint32Value (const uint32_t nEntryID);
		uint16_t getUint16Value (const uint32_t nEntryID);
		uint8_t getUint8Value (const uint32_t nEntryID);

	};

	template<typename T> class ioModuleAccess {

		private:
		T * m_Module;

		public:

		ioModuleAccess (CEnvironment * pEnvironment, const std::string & sModuleName)
			: m_Module (nullptr)
		{
			auto pModule = pEnvironment->findModule (sModuleName, true);
			if (pModule->isActive ()) {
				auto pCastedModule = dynamic_cast<T *> (pModule);

				if (pCastedModule != nullptr)
				{
					m_Module = pCastedModule;
				} else
				{
					throw CException (eErrorCode::INVALIDMODULETYPE, "invalid module type: " + sModuleName);
				}

			} else
				throw CException (eErrorCode::MODULENOTACTIVE, "module not active: " + sModuleName);

		}

		virtual ~ioModuleAccess  ()
		{
		}

		T& operator* ()
		{
			return *m_Module;
		}

		T* operator-> ()
		{
			return m_Module;
		}

	};

}

#endif // __FRAMEWORK_HPP
```

#### Framework.cpp
```cpp
/*++

Copyright (C) 2024 Institute for Machine Tools and Industrial Management
TUM School of Engineering and Design
Technical University of Munich

All rights reserved.

Redistribution and use in source and binary forms, with or without
modification, are permitted provided that the following conditions are met:
	* Redistributions of source code must retain the above copyright
	  notice, this list of conditions and the following disclaimer.
	* Redistributions in binary form must reproduce the above copyright
	  notice, this list of conditions and the following disclaimer in the
	  documentation and/or other materials provided with the distribution.
	* Neither the name of the Technical University of Munich nor the
	  names of its contributors may be used to endorse or promote products
	  derived from this software without specific prior written permission.

THIS SOFTWARE IS PROVIDED BY THE COPYRIGHT HOLDERS AND CONTRIBUTORS "AS IS" AND
ANY EXPRESS OR IMPLIED WARRANTIES, INCLUDING, BUT NOT LIMITED TO, THE IMPLIED
WARRANTIES OF MERCHANTABILITY AND FITNESS FOR A PARTICULAR PURPOSE ARE
DISCLAIMED. IN NO EVENT SHALL TECHNICAL UNIVERSITY OF MUNICH BE LIABLE FOR ANY
DIRECT, INDIRECT, INCIDENTAL, SPECIAL, EXEMPLARY, OR CONSEQUENTIAL DAMAGES
(INCLUDING, BUT NOT LIMITED TO, PROCUREMENT OF SUBSTITUTE GOODS OR SERVICES;
LOSS OF USE, DATA, OR PROFITS; OR BUSINESS INTERRUPTION) HOWEVER CAUSED AND
ON ANY THEORY OF LIABILITY, WHETHER IN CONTRACT, STRICT LIABILITY, OR TORT
(INCLUDING NEGLIGENCE OR OTHERWISE) ARISING IN ANY WAY OUT OF THE USE OF THIS
SOFTWARE, EVEN IF ADVISED OF THE POSSIBILITY OF SUCH DAMAGE.

*/

#include "Framework.hpp"
#include "SignalHandler.hpp"
#include "Utils.hpp"
#include "Journal.hpp"
#include <stdint.h>

namespace BuRCPP {

	CException::CException (eErrorCode code, const std::string & sMessage)
		: m_Code (code), m_sMessage (sMessage)
	{
	}

	eErrorCode CException::getCode () const
	{
		return m_Code;
	}

	const char * CException::getMessage () const
	{
		return m_sMessage.c_str ();
	}

CModule::CModule (const std::string & sName)
	: m_sName (sName), m_bJournalIsRegistering (false)
{
}

CModule::~CModule ()
{
}

std::string CModule::getName ()
{
	return m_sName;
}

void CModule::handleCyclic ()
{
}

void CModule::setJournal (std::shared_ptr<CJournal> pJournal, uint32_t nJournalGroupID)
{
	if (pJournal.get () == nullptr)
		throw CException (eErrorCode::INVALIDPARAM, "invalid journal parameter");
	if (m_bJournalIsRegistering)
		throw CException (eErrorCode::JOURNALALREADYREGISTERING, "journal is already registering");

	m_pJournal = pJournal;
	m_nJournalGroupID = nJournalGroupID;

	m_pJournal->registerGroup (nJournalGroupID, m_sName);

	m_bJournalIsRegistering = true;
	try {
		onRegisterJournal ();
	}
	catch (...) {
		m_bJournalIsRegistering = false;
		throw;
	}
}

void CModule::onRegisterJournal ()
{
}

void CModule::onUpdateJournal ()
{
}

void CModule::registerIntegerValue (const std::string & sEntryName,const uint32_t nEntryID, int64_t nMinValue, int64_t nMaxValue)
{
	if (m_pJournal.get () == nullptr)
		throw CException (eErrorCode::JOURNALNOTSET, "journal is not set");
	if (!m_bJournalIsRegistering)
		throw CException (eErrorCode::JOURNALISNOTREGISTERING, "journal is not registering");

	m_pJournal->registerIntegerValue (sEntryName, m_nJournalGroupID, nEntryID, nMinValue, nMaxValue);
}

void CModule::registerBoolValue (const std::string & sEntryName,const uint32_t nEntryID)
{
	if (m_pJournal.get () == nullptr)
		throw CException (eErrorCode::JOURNALNOTSET, "journal is not set");
	if (!m_bJournalIsRegistering)
		throw CException (eErrorCode::JOURNALISNOTREGISTERING, "journal is not registering");

	m_pJournal->registerBoolValue (sEntryName, m_nJournalGroupID, nEntryID);
}

void CModule::registerDoubleValue (const std::string & sEntryName,const uint32_t nEntryID, double dMinValue, double dMaxValue, int64_t nQuantizationSteps)
{
	if (m_pJournal.get () == nullptr)
		throw CException (eErrorCode::JOURNALNOTSET, "journal is not set");
	if (!m_bJournalIsRegistering)
		throw CException (eErrorCode::JOURNALISNOTREGISTERING, "journal is not registering");

	m_pJournal->registerDoubleValue (sEntryName, m_nJournalGroupID, nEntryID, dMinValue, dMaxValue, nQuantizationSteps);

}

void CModule::registerUInt8Value (const std::string & sEntryName,const uint32_t nEntryID)
{
	registerIntegerValue (sEntryName, nEntryID, 0, UINT8_MAX);
}

void CModule::registerUInt16Value (const std::string & sEntryName,const uint32_t nEntryID)
{
	registerIntegerValue (sEntryName, nEntryID, 0, UINT16_MAX);
}

void CModule::registerUInt32Value (const std::string & sEntryName,const uint32_t nEntryID)
{
	registerIntegerValue (sEntryName, nEntryID, 0, UINT32_MAX);
}

void CModule::registerInt8Value (const std::string & sEntryName,const uint32_t nEntryID)
{
	registerIntegerValue (sEntryName, nEntryID, INT8_MIN, INT8_MAX);
}

void CModule::registerInt16Value (const std::string & sEntryName,const uint32_t nEntryID)
{
	registerIntegerValue (sEntryName, nEntryID, INT16_MIN, INT16_MAX);
}

void CModule::registerInt32Value (const std::string & sEntryName,const uint32_t nEntryID)
{
	registerIntegerValue (sEntryName, nEntryID, INT32_MIN, INT32_MAX);
}

void CModule::setIntegerValue (const uint32_t nEntryID, int64_t nValue)
{
	if (m_pJournal.get () == nullptr)
		throw CException (eErrorCode::JOURNALNOTSET, "journal is not set");

	m_pJournal->setIntegerValue (m_nJournalGroupID, nEntryID, nValue);
}

void CModule::setBoolValue (const uint32_t nEntryID, bool bValue)
{
	if (m_pJournal.get () == nullptr)
		throw CException (eErrorCode::JOURNALNOTSET, "journal is not set");

	m_pJournal->setBoolValue (m_nJournalGroupID, nEntryID, bValue);
}

void CModule::setDoubleValue (const uint32_t nEntryID, double dValue)
{
	if (m_pJournal.get () == nullptr)
		throw CException (eErrorCode::JOURNALNOTSET, "journal is not set");

	m_pJournal->setDoubleValue (m_nJournalGroupID, nEntryID, dValue);
}

CIOModule::CIOModule (const std::string & sName)
	: CModule (sName)
{
}

CIOModule::~CIOModule ()
{
}

CAxisModule::CAxisModule (const std::string & sName)
	: CModule (sName)
{
}

CAxisModule::~CAxisModule ()
{
}

void CAxisModule::setPowerOn ()
{
	setPower (true);
}

void CAxisModule::setPowerOff ()
{
	setPower (false);
}

CEnvironment::CEnvironment (CStateHandler * pStateHandler)
	: m_pStateHandler (pStateHandler), m_pNextState (nullptr)
{
	if (pStateHandler == nullptr)
		throw CException (eErrorCode::INVALIDPARAM, "invalid state handler parameter");
}

CEnvironment::~CEnvironment ()
{
}

CState * CEnvironment::getNextState ()
{
	return m_pNextState;
}

void CEnvironment::setNextState (const std::string & sNextState)
{
	CState * pState = m_pStateHandler->findState (sNextState);
	if (pState == nullptr)
		throw CException (eErrorCode::STATENOTFOUND, "state has not been found: " + sNextState);

	m_pNextState = pState;
}

CModule * CEnvironment::findModule (const std::string & sName, bool bFailIfNotExist)
{
	auto pModule = m_pStateHandler->findModule (sName);
	if (pModule == nullptr) {
		if (bFailIfNotExist)
			throw CException (eErrorCode::MODULENOTFOUND, "module has not been found: " + sName);
	}

	return pModule;

}

CSignalProcessingInstance * CEnvironment::checkSignal (const std::string & sName)
{
	auto pSignalHandler = m_pStateHandler->getSignalHandler();
	if (pSignalHandler != nullptr) {
		return pSignalHandler->checkSignal (sName);
	}

	return nullptr;
}

void CEnvironment::setIntegerValue (const uint32_t nEntryID, int64_t nValue)
{
	m_pStateHandler->setIntegerValue (nEntryID, nValue);
}

void CEnvironment::setBoolValue (const uint32_t nEntryID, bool bValue)
{
	m_pStateHandler->setBoolValue (nEntryID, bValue);
}

void CEnvironment::setDoubleValue (const uint32_t nEntryID, double dValue)
{
	m_pStateHandler->setDoubleValue (nEntryID, dValue);
}

bool CEnvironment::getBoolValue (const uint32_t nEntryID)
{
	return m_pStateHandler->getBoolValue (nEntryID);
}

double CEnvironment::getDoubleValue (const uint32_t nEntryID)
{
	return m_pStateHandler->getDoubleValue (nEntryID);
}

int64_t CEnvironment::getInt64Value (const uint32_t nEntryID)
{
	return m_pStateHandler->getInt64Value (nEntryID);
}

int32_t CEnvironment::getInt32Value (const uint32_t nEntryID)
{
	return m_pStateHandler->getInt32Value (nEntryID);
}

int16_t CEnvironment::getInt16Value (const uint32_t nEntryID)
{
	return m_pStateHandler->getInt16Value (nEntryID);
}

int8_t CEnvironment::getInt8Value (const uint32_t nEntryID)
{
	return m_pStateHandler->getInt8Value (nEntryID);
}

uint64_t CEnvironment::getUint64Value (const uint32_t nEntryID)
{
	return m_pStateHandler->getUint64Value (nEntryID);
}

uint32_t CEnvironment::getUint32Value (const uint32_t nEntryID)
{
	return m_pStateHandler->getUint32Value (nEntryID);
}

uint16_t CEnvironment::getUint16Value (const uint32_t nEntryID)
{
	return m_pStateHandler->getUint32Value (nEntryID);
}

uint8_t CEnvironment::getUint8Value (const uint32_t nEntryID)
{
	return m_pStateHandler->getUint8Value (nEntryID);
}

CState::CState ()
{
}

CState::~CState ()
{
}

CModuleHandler::CModuleHandler (std::shared_ptr<CJournal> pJournal)
		: m_pJournal (pJournal)
{
	if (pJournal.get () == nullptr)
		throw CException (eErrorCode::INVALIDPARAM, "invalid journal parameter");

}

CModuleHandler::~CModuleHandler ()
{
}

void CModuleHandler::handleModules ()
{
	for (auto iIterator : m_Modules)
		iIterator.second->handleCyclic ();
	for (auto iIterator : m_Modules)
		iIterator.second->onUpdateJournal ();
}

CModule * CModuleHandler::findModule (const std::string & sName)
{
	auto iIter = m_Modules.find (sName);
	if (iIter != m_Modules.end ())
		return iIter->second.get();

	return nullptr;
}

void CModuleHandler::registerModule (std::shared_ptr<CModule> pModule, uint32_t nJournalGroupID)
{
	if (pModule.get () == nullptr)
		throw CException (eErrorCode::INVALIDPARAM, "invalid module parameter");

	std::string sName = pModule->getName ();
	if (findModule (sName) != nullptr)
		throw CException (eErrorCode::MODULEALREADYEXISTS, "module already exists");

	m_Modules.insert (std::make_pair (sName, pModule));

	pModule->setJournal (m_pJournal, nJournalGroupID);

}

CStateHandler::CStateHandler (std::shared_ptr<CJournal> pJournal, const std::string & sName, std::shared_ptr<CModuleHandler> pModuleHandler, uint32_t nJournalGroupID)
	: m_pCurrentState (nullptr), m_pStateNameDebug (nullptr), m_nStateNameDebugLength (0), m_pJournal (pJournal), m_nJournalGroupID (nJournalGroupID), m_sName (sName), m_pModuleHandler (pModuleHandler)
{
	if (pJournal.get () == nullptr)
		throw CException (eErrorCode::INVALIDPARAM, "invalid journal parameter");

	if (pModuleHandler.get () == nullptr)
		throw CException (eErrorCode::INVALIDPARAM, "invalid module handler parameter");

	m_pSignalHandler = std::make_shared<CSignalHandler> (pJournal->getSystemInfo ());
	pJournal->registerGroup (nJournalGroupID, getName ());

}

CStateHandler::~CStateHandler()
{
}

std::string CStateHandler::getName ()
{
	return m_sName;
}

CState * CStateHandler::findState (const std::string & sName) {

	auto iIter = m_States.find (sName);
	if (iIter != m_States.end ())
		return iIter->second.get();

	return nullptr;

}

void CStateHandler::addState (std::shared_ptr<CState> pState)
{

	if (pState.get () == nullptr)
		throw CException (eErrorCode::INVALIDPARAM, "invalid state parameter");

	std::string sName = pState->getName ();
	if (findState (sName) != nullptr)
		throw CException (eErrorCode::STATEALREADYEXISTS, "state already exists");

	m_States.insert (std::make_pair (sName, pState));

	if (m_pCurrentState == nullptr)
		m_pCurrentState = pState.get();

}

void CStateHandler::setCurrentState (CState * pState)
{
	if (pState == nullptr)
		throw CException (eErrorCode::INVALIDPARAM, "invalid state parameter");

	m_pCurrentState = pState;

}

CState * CStateHandler::getCurrentState ()
{
	return m_pCurrentState;
}

CModule * CStateHandler::findModule (const std::string & sName)
{
	return m_pModuleHandler->findModule (sName);
}

CSignalHandler* CStateHandler::getSignalHandler ()
{
	return m_pSignalHandler.get ();
}

std::shared_ptr<CSignalDefinition> CStateHandler::registerSignal (const std::string & sName, const uint32_t nQueueSize, const uint32_t nLifetimeInMilliseconds)
{
	return m_pSignalHandler->registerSignal (sName, nQueueSize, nLifetimeInMilliseconds);
}

void CStateHandler::onRegister ()
{
	// Build Signal Handler Instances
	m_pSignalHandler->buildInstances ();
}

void CStateHandler::setDebugVariables (char * pStateNameDebug, uint32_t nStateNameDebugLength)
{
	m_pStateNameDebug = pStateNameDebug;
	m_nStateNameDebugLength = nStateNameDebugLength;
}

void CStateHandler::writeDebugInformation ()
{
	if ((m_pStateNameDebug != nullptr) && (m_nStateNameDebugLength > 0)) {

		if (m_pCurrentState != nullptr) {

			std::string sStateName = m_pCurrentState->getName();
			CUtils::writeStringVariable (sStateName, m_pStateNameDebug, m_nStateNameDebugLength);

		} else {

			CUtils::writeStringVariable ("<null>", m_pStateNameDebug, m_nStateNameDebugLength);

		}

	}
}

void CStateHandler::registerIntegerValue (const std::string & sEntryName,const uint32_t nEntryID, int64_t nMinValue, int64_t nMaxValue)
{
	m_pJournal->registerIntegerValue (sEntryName, m_nJournalGroupID, nEntryID, nMinValue, nMaxValue);
}

void CStateHandler::registerBoolValue (const std::string & sEntryName,const uint32_t nEntryID)
{
	m_pJournal->registerBoolValue (sEntryName, m_nJournalGroupID, nEntryID);
}

void CStateHandler::registerDoubleValue (const std::string & sEntryName,const uint32_t nEntryID, double dMinValue, double dMaxValue, int64_t nQuantizationSteps)
{
	m_pJournal->registerDoubleValue (sEntryName, m_nJournalGroupID, nEntryID, dMinValue, dMaxValue, nQuantizationSteps);
}

void CStateHandler::setIntegerValue (const uint32_t nEntryID, int64_t nValue)
{
	m_pJournal->setIntegerValue (m_nJournalGroupID, nEntryID, nValue );
}

void CStateHandler::setBoolValue (const uint32_t nEntryID, bool bValue)
{
	m_pJournal->setBoolValue (m_nJournalGroupID, nEntryID, bValue );
}

void CStateHandler::setDoubleValue (const uint32_t nEntryID, double dValue)
{
	m_pJournal->setDoubleValue (m_nJournalGroupID, nEntryID, dValue );
}

bool CStateHandler::getBoolValue (const uint32_t nEntryID)
{
	return m_pJournal->getBoolValue (m_nJournalGroupID, nEntryID);
}

double CStateHandler::getDoubleValue (const uint32_t nEntryID)
{
	return m_pJournal->getDoubleValue (m_nJournalGroupID, nEntryID);
}

int64_t CStateHandler::getInt64Value (const uint32_t nEntryID)
{
	return m_pJournal->getInt64Value (m_nJournalGroupID, nEntryID);
}

int32_t CStateHandler::getInt32Value (const uint32_t nEntryID)
{
	return m_pJournal->getInt32Value (m_nJournalGroupID, nEntryID);
}

int16_t CStateHandler::getInt16Value (const uint32_t nEntryID)
{
	return m_pJournal->getInt16Value (m_nJournalGroupID, nEntryID);
}

int8_t CStateHandler::getInt8Value (const uint32_t nEntryID)
{
	return m_pJournal->getInt8Value (m_nJournalGroupID, nEntryID);
}

uint64_t CStateHandler::getUint64Value (const uint32_t nEntryID)
{
	return m_pJournal->getUint64Value (m_nJournalGroupID, nEntryID);
}

uint32_t CStateHandler::getUint32Value (const uint32_t nEntryID)
{
	return m_pJournal->getUint32Value (m_nJournalGroupID, nEntryID);
}

uint16_t CStateHandler::getUint16Value (const uint32_t nEntryID)
{
	return m_pJournal->getUint16Value (m_nJournalGroupID, nEntryID);
}

uint8_t CStateHandler::getUint8Value (const uint32_t nEntryID)
{
	return m_pJournal->getUint8Value (m_nJournalGroupID, nEntryID);
}

void CStateHandler::releaseExpiredSignals ()
{
		m_pSignalHandler->releaseExpiredSignals ();
}

}
```

#### SystemInfo.hpp
```cpp
/*++

Copyright (C) 2024 Institute for Machine Tools and Industrial Management
TUM School of Engineering and Design
Technical University of Munich

All rights reserved.

Redistribution and use in source and binary forms, with or without
modification, are permitted provided that the following conditions are met:
	* Redistributions of source code must retain the above copyright
	  notice, this list of conditions and the following disclaimer.
	* Redistributions in binary form must reproduce the above copyright
	  notice, this list of conditions and the following disclaimer in the
	  documentation and/or other materials provided with the distribution.
	* Neither the name of the Technical University of Munich nor the
	  names of its contributors may be used to endorse or promote products
	  derived from this software without specific prior written permission.

THIS SOFTWARE IS PROVIDED BY THE COPYRIGHT HOLDERS AND CONTRIBUTORS "AS IS" AND
ANY EXPRESS OR IMPLIED WARRANTIES, INCLUDING, BUT NOT LIMITED TO, THE IMPLIED
WARRANTIES OF MERCHANTABILITY AND FITNESS FOR A PARTICULAR PURPOSE ARE
DISCLAIMED. IN NO EVENT SHALL TECHNICAL UNIVERSITY OF MUNICH BE LIABLE FOR ANY
DIRECT, INDIRECT, INCIDENTAL, SPECIAL, EXEMPLARY, OR CONSEQUENTIAL DAMAGES
(INCLUDING, BUT NOT LIMITED TO, PROCUREMENT OF SUBSTITUTE GOODS OR SERVICES;
LOSS OF USE, DATA, OR PROFITS; OR BUSINESS INTERRUPTION) HOWEVER CAUSED AND
ON ANY THEORY OF LIABILITY, WHETHER IN CONTRACT, STRICT LIABILITY, OR TORT
(INCLUDING NEGLIGENCE OR OTHERWISE) ARISING IN ANY WAY OUT OF THE USE OF THIS
SOFTWARE, EVEN IF ADVISED OF THE POSSIBILITY OF SUCH DAMAGE.

*/

#ifndef __SYSTEMINFO_HPP
#define __SYSTEMINFO_HPP

#include "Framework.hpp"

namespace BuRCPP {

	class CSystemInfo {
		protected:

			uint64_t m_nStartSystemTime;
			uint64_t m_nSystemTimeCycle;
			uint32_t m_nCurrentSystemTimeRegister;

		public:

		CSystemInfo ();
		virtual ~CSystemInfo ();

		uint64_t getSystemTimeInMicroseconds ();

		uint64_t getSystemTimeInMilliseconds ();

		void handleCyclic ();

	};

}

#endif //__SYSTEMINFO_HPP
```

#### SystemInfo.cpp
```cpp
/*++

Copyright (C) 2024 Institute for Machine Tools and Industrial Management
TUM School of Engineering and Design
Technical University of Munich

All rights reserved.

Redistribution and use in source and binary forms, with or without
modification, are permitted provided that the following conditions are met:
	* Redistributions of source code must retain the above copyright
	  notice, this list of conditions and the following disclaimer.
	* Redistributions in binary form must reproduce the above copyright
	  notice, this list of conditions and the following disclaimer in the
	  documentation and/or other materials provided with the distribution.
	* Neither the name of the Technical University of Munich nor the
	  names of its contributors may be used to endorse or promote products
	  derived from this software without specific prior written permission.

THIS SOFTWARE IS PROVIDED BY THE COPYRIGHT HOLDERS AND CONTRIBUTORS "AS IS" AND
ANY EXPRESS OR IMPLIED WARRANTIES, INCLUDING, BUT NOT LIMITED TO, THE IMPLIED
WARRANTIES OF MERCHANTABILITY AND FITNESS FOR A PARTICULAR PURPOSE ARE
DISCLAIMED. IN NO EVENT SHALL TECHNICAL UNIVERSITY OF MUNICH BE LIABLE FOR ANY
DIRECT, INDIRECT, INCIDENTAL, SPECIAL, EXEMPLARY, OR CONSEQUENTIAL DAMAGES
(INCLUDING, BUT NOT LIMITED TO, PROCUREMENT OF SUBSTITUTE GOODS OR SERVICES;
LOSS OF USE, DATA, OR PROFITS; OR BUSINESS INTERRUPTION) HOWEVER CAUSED AND
ON ANY THEORY OF LIABILITY, WHETHER IN CONTRACT, STRICT LIABILITY, OR TORT
(INCLUDING NEGLIGENCE OR OTHERWISE) ARISING IN ANY WAY OUT OF THE USE OF THIS
SOFTWARE, EVEN IF ADVISED OF THE POSSIBILITY OF SUCH DAMAGE.

*/

#include "SystemInfo.hpp"

// Raw Registers

namespace BuRCPP {

	CSystemInfo::CSystemInfo ()
		: m_nSystemTimeCycle (0),
		m_nCurrentSystemTimeRegister (0),
		m_nStartSystemTime (0)
	{
		m_nStartSystemTime = IOMapping_PLC.SystemTime;
	}

	CSystemInfo::~CSystemInfo ()
	{
	}

	uint64_t CSystemInfo::getSystemTimeInMicroseconds ()
	{
		handleCyclic ();
		return (( m_nSystemTimeCycle << 32) | (uint64_t) m_nCurrentSystemTimeRegister) - m_nStartSystemTime;
	}

	uint64_t CSystemInfo::getSystemTimeInMilliseconds ()
	{
		return getSystemTimeInMicroseconds () / 1000;
	}

	void CSystemInfo::handleCyclic ()
	{
		uint32_t nNewRegister = IOMapping_PLC.SystemTime;
		if (nNewRegister < m_nCurrentSystemTimeRegister)
			m_nSystemTimeCycle ++;
		m_nCurrentSystemTimeRegister = nNewRegister;
	}

}
```

#### TcpServer.hpp
```cpp
/*++

Copyright (C) 2024 Institute for Machine Tools and Industrial Management
TUM School of Engineering and Design
Technical University of Munich

All rights reserved.

Redistribution and use in source and binary forms, with or without
modification, are permitted provided that the following conditions are met:
	* Redistributions of source code must retain the above copyright
	  notice, this list of conditions and the following disclaimer.
	* Redistributions in binary form must reproduce the above copyright
	  notice, this list of conditions and the following disclaimer in the
	  documentation and/or other materials provided with the distribution.
	* Neither the name of the Technical University of Munich nor the
	  names of its contributors may be used to endorse or promote products
	  derived from this software without specific prior written permission.

THIS SOFTWARE IS PROVIDED BY THE COPYRIGHT HOLDERS AND CONTRIBUTORS "AS IS" AND
ANY EXPRESS OR IMPLIED WARRANTIES, INCLUDING, BUT NOT LIMITED TO, THE IMPLIED
WARRANTIES OF MERCHANTABILITY AND FITNESS FOR A PARTICULAR PURPOSE ARE
DISCLAIMED. IN NO EVENT SHALL TECHNICAL UNIVERSITY OF MUNICH BE LIABLE FOR ANY
DIRECT, INDIRECT, INCIDENTAL, SPECIAL, EXEMPLARY, OR CONSEQUENTIAL DAMAGES
(INCLUDING, BUT NOT LIMITED TO, PROCUREMENT OF SUBSTITUTE GOODS OR SERVICES;
LOSS OF USE, DATA, OR PROFITS; OR BUSINESS INTERRUPTION) HOWEVER CAUSED AND
ON ANY THEORY OF LIABILITY, WHETHER IN CONTRACT, STRICT LIABILITY, OR TORT
(INCLUDING NEGLIGENCE OR OTHERWISE) ARISING IN ANY WAY OUT OF THE USE OF THIS
SOFTWARE, EVEN IF ADVISED OF THE POSSIBILITY OF SUCH DAMAGE.

*/

#ifndef __TCPSERVER_HPP
#define __TCPSERVER_HPP

#include "Framework.hpp"
#include "TcpPacketHandler.hpp"
#include <list>
#include <vector>

#define TCPMINBUFFERSIZE 1024
#define TCPMAXBUFFERSIZE (16*1024*1024)

namespace BuRCPP {

	class CTcpServerImpl;
	class CTcpConnectionImpl;

	enum class eTcpServer_State : int32_t
	{
		UNKNOWN = 0,
		INACTIVE = 1,
		INIT	 = 2,
		INITIALIZING = 3,
		LISTENING	= 4,
		CLOSINGCONNECTION = 5,
		ERROR =	6
	};

	enum class eTcpConnectionRecv_State : int32_t
	{
		UNKNOWN = 0,
		INACTIVE = 1,
		WAITINGFORDATA = 2,
		RESETCONNECTION = 3,
		CLOSINGCONNECTION = 4,
		ERROR =	6
	};

	enum class eTcpConnectionSend_State : int32_t
	{
		UNKNOWN = 0,
		INACTIVE = 1,
		WAITINGFORDATA = 2,
		CLOSINGCONNECTION = 4,
		SENDING = 5,
		ERROR =	6
	};

	class CTcpConnection {
		protected:
			std::shared_ptr<CTcpConnectionImpl> m_pImpl;
			uint32_t m_ClientIdent;
			eTcpConnectionRecv_State m_RecvState;
			eTcpConnectionSend_State m_SendState;

			std::vector<uint8_t> m_ReceiveBuffer;
			std::vector<uint8_t> m_SendBuffer1;
			std::vector<uint8_t> m_SendBuffer2;

			uint8_t * m_pSendBufferInProcess;
			uint8_t * m_pSendBufferNextInQueue;
			uint32_t m_SendBufferInProcessSize;
			uint32_t m_SendBufferNextInQueueSize;
			uint32_t m_SendBufferMemorySize;

			CTcpPacketRegistry* m_pPacketRegistry;

			CTcpPacketResponse m_TempResponse;

			uint32_t m_LastError;

		public:

		CTcpConnection (uint32_t nReceiveBufferSize, uint32_t nSendBufferSize, CTcpPacketRegistry* pPacketRegistry);
		virtual ~CTcpConnection ();

		void initialize (uint32_t clientIdent);

		void handleCyclic ();

		bool canSendData (uint32_t nByteCount);

		void sendData (uint8_t * pBytes, uint32_t nByteCount);

	};

	class CTcpServer {

		protected:
		std::shared_ptr<CTcpServerImpl> m_pImpl;
		std::list<std::shared_ptr<CTcpConnection>> m_InactiveConnections;
		std::list<std::shared_ptr<CTcpConnection>> m_ActiveConnections;
		std::shared_ptr<CTcpPacketRegistry> m_PacketRegistry;

		eTcpServer_State m_State;
		uint32_t m_Port;
		uint32_t m_MaxConnections;
		uint32_t m_LastError;

		bool enableConnection (uint32_t nClientIdent);

		public:

		CTcpServer (uint32_t port, uint32_t maxConnections, uint32_t nPacketSignature);
		virtual ~CTcpServer();

		virtual bool serverRunning ();
		virtual bool clientConnected ();

		virtual void startServer ();
		virtual void stopServer ();

		virtual void handleServer ();

		void registerPacketHandler (std::shared_ptr<CTcpPacketHandler> pPacketHandler);

		void * getFunctionBlockOpen ();
		void * getFunctionBlockClose ();
		void * getFunctionBlockServer ();

		CTcpPacketRegistry * getPacketRegistry ();

	};

}

#endif
```

#### TcpServer.cpp
```cpp
/*++

Copyright (C) 2024 Institute for Machine Tools and Industrial Management
TUM School of Engineering and Design
Technical University of Munich

All rights reserved.

Redistribution and use in source and binary forms, with or without
modification, are permitted provided that the following conditions are met:
	* Redistributions of source code must retain the above copyright
	  notice, this list of conditions and the following disclaimer.
	* Redistributions in binary form must reproduce the above copyright
	  notice, this list of conditions and the following disclaimer in the
	  documentation and/or other materials provided with the distribution.
	* Neither the name of the Technical University of Munich nor the
	  names of its contributors may be used to endorse or promote products
	  derived from this software without specific prior written permission.

THIS SOFTWARE IS PROVIDED BY THE COPYRIGHT HOLDERS AND CONTRIBUTORS "AS IS" AND
ANY EXPRESS OR IMPLIED WARRANTIES, INCLUDING, BUT NOT LIMITED TO, THE IMPLIED
WARRANTIES OF MERCHANTABILITY AND FITNESS FOR A PARTICULAR PURPOSE ARE
DISCLAIMED. IN NO EVENT SHALL TECHNICAL UNIVERSITY OF MUNICH BE LIABLE FOR ANY
DIRECT, INDIRECT, INCIDENTAL, SPECIAL, EXEMPLARY, OR CONSEQUENTIAL DAMAGES
(INCLUDING, BUT NOT LIMITED TO, PROCUREMENT OF SUBSTITUTE GOODS OR SERVICES;
LOSS OF USE, DATA, OR PROFITS; OR BUSINESS INTERRUPTION) HOWEVER CAUSED AND
ON ANY THEORY OF LIABILITY, WHETHER IN CONTRACT, STRICT LIABILITY, OR TORT
(INCLUDING NEGLIGENCE OR OTHERWISE) ARISING IN ANY WAY OUT OF THE USE OF THIS
SOFTWARE, EVEN IF ADVISED OF THE POSSIBILITY OF SUCH DAMAGE.

*/

#include "TcpServer.hpp"

#include <bur/plctypes.h>

#ifdef _DEFAULT_INCLUDES
#include <AsDefault.h>
#endif

#include <string.h>

namespace BuRCPP
{

	class CTcpServerImpl
	{
		private:

		TcpOpen_typ m_TcpOpen;
		TcpServer_typ m_TcpServer;
		TcpClose_typ m_TcpClose;

		char m_ServerClientAddress[80];

		public:

		CTcpServerImpl () {
			memset ((void*) &m_TcpOpen, 0, sizeof (m_TcpOpen));
			memset ((void*) &m_TcpServer, 0, sizeof (m_TcpServer));
			memset ((void*) &m_TcpClose, 0, sizeof (m_TcpClose));

		}

		void handleCyclic ()
		{
			TcpOpen(&m_TcpOpen);
			TcpServer(&m_TcpServer);
			TcpClose(&m_TcpClose);
		}

		void * getFunctionBlockOpen ()
		{
			return &m_TcpOpen;
		}

		void * getFunctionBlockClose ()
		{
			return &m_TcpClose;
		}

		void * getFunctionBlockServer ()
		{
			return &m_TcpServer;
		}

		void initialiseTCP (uint32_t nPort)
		{
			m_TcpOpen.pIfAddr = 0; // Take IP Adress vom ETH Configuration
			m_TcpOpen.port = nPort;
			m_TcpOpen.options = 0;
			m_TcpOpen.enable = 1;
		}

		bool tcpOpenIsBusy ()
		{
			return (tcpOpenErrorCode () == 65535);
		}

		bool tcpOpenIsFinished ()
		{
			return (tcpOpenErrorCode () == 0);
		}

		uint32_t tcpOpenErrorCode ()
		{
			return m_TcpOpen.status;
		}

		uint32_t tcpOpenIdent ()
		{
			return m_TcpOpen.ident;
		}

		uint32_t tcpListenClientIdent ()
		{
			return m_TcpServer.identclnt;
		}

		bool tcpListenClientConnected ()
		{
			return (tcpListenErrorCode () == 0);
		}

		bool tcpListenIsBusy ()
		{
			return (tcpListenErrorCode() == 65535);
		}

		uint32_t tcpListenErrorCode ()
		{
			return m_TcpServer.status;
		}

		bool tcpCloseFinished ()
		{
			return (tcpCloseErrorCode () == 0);
		}

		bool tcpCloseIsBusy ()
		{
			return (tcpCloseErrorCode() == 65535);
		}

		uint32_t tcpCloseErrorCode ()
		{
			return m_TcpClose.status;
		}

		void listenOnSocket (uint32_t nSocketIdent, uint32_t nMaxConnections)
		{
			//Configure TCP Server
			m_TcpServer.enable = 1;
			m_TcpServer.ident = nSocketIdent;
			m_TcpServer.backlog = nMaxConnections;
			m_TcpServer.pIpAddr = (UDINT)&m_ServerClientAddress;
		}

		void closeClientConnection (uint32_t nClientIdent)
		{
			m_TcpClose.enable = 1;
			m_TcpClose.ident = nClientIdent;
			m_TcpClose.how = 0;

		}

		void resetClose ()
		{
			m_TcpClose.enable = 0;
		}

	};

	class CTcpConnectionImpl
	{
		private:

			TcpRecv_typ m_TcpReceive;
			TcpSend_typ m_TcpSend;
			TcpClose_typ m_TcpClose;

		public:

			CTcpConnectionImpl () {
				resetFunctionBlocks ();

			}

			virtual ~CTcpConnectionImpl ()
			{
			}

			void resetFunctionBlocks ()
			{
			memset ((void*) &m_TcpReceive, 0, sizeof (m_TcpReceive));
			memset ((void*) &m_TcpSend, 0, sizeof (m_TcpSend));
			memset ((void*) &m_TcpClose, 0, sizeof (m_TcpClose));
		}

		void handleCyclic ()
		{
			TcpRecv(&m_TcpReceive);
			TcpSend(&m_TcpSend);
		}

		void * getFunctionBlockClose ()
		{
			return &m_TcpClose;
		}

		void * getFunctionBlockSend ()
		{
			return &m_TcpSend;
		}

		void * getFunctionBlockRecv ()
		{
			return &m_TcpReceive;
		}

		void initReceive (uint32_t nClientIdent, void * pBuffer, uint32_t nBufferSize)
		{
			m_TcpReceive.enable = 1;
			m_TcpReceive.ident = nClientIdent;
			m_TcpReceive.flags = 0;
			m_TcpReceive.datamax = nBufferSize;
			m_TcpReceive.pData = (UDINT) pBuffer;
		}

		void resetReceive ()
		{
			memset ((void*) &m_TcpReceive, 0, sizeof (m_TcpReceive));
		}

		bool tcpRecvIsFinished ()
		{
			return (tcpRecvErrorCode () == 0);
		}

		bool tcpRecvIsBusy ()
		{
			return (tcpRecvErrorCode () == 65535) || (tcpRecvErrorCode () == 32605);
		}

		uint32_t tcpRecvErrorCode ()
		{
			return m_TcpReceive.status;
		}

		uint32_t tcpBytesReceived ()
		{
			return m_TcpReceive.recvlen;
		}

		void initSend (uint32_t nClientIdent, void * pBuffer, uint32_t nBufferSize)
		{
			m_TcpSend.enable = 1;
			m_TcpSend.ident = nClientIdent;
			m_TcpSend.datalen = nBufferSize;
			m_TcpSend.flags = 0;
			m_TcpSend.pData = (UDINT) pBuffer;
		}

		void resetSend ()
		{
			memset ((void*) &m_TcpSend, 0, sizeof (m_TcpSend));
		}

		bool tcpSendIsFinished ()
		{
			return (tcpSendErrorCode () == 0);
		}

		bool tcpSendIsBusy ()
		{
			return (tcpSendErrorCode () == 65535);
		}

		uint32_t tcpSendErrorCode ()
		{
			return m_TcpSend.status;
		}

		uint32_t tcpBytesSent ()
		{
			return m_TcpSend.sentlen;
		}

	};

	CTcpConnection::CTcpConnection (uint32_t nReceiveBufferSize, uint32_t nSendBufferSize, CTcpPacketRegistry* pPacketRegistry)
		: m_SendState (eTcpConnectionSend_State::INACTIVE),
		m_RecvState (eTcpConnectionRecv_State::INACTIVE),
		m_ClientIdent (0), m_LastError (0),
		m_SendBufferInProcessSize (0),
		m_SendBufferNextInQueueSize (0),
		m_SendBufferMemorySize (nSendBufferSize),
		m_pPacketRegistry (pPacketRegistry)

	{
		if (pPacketRegistry == nullptr)
			throw CException (eErrorCode::INVALIDPARAM, "invalid packet registry.");
		if ((nReceiveBufferSize < TCPMINBUFFERSIZE) || (nReceiveBufferSize > TCPMAXBUFFERSIZE))
			throw CException (eErrorCode::INVALIDTCPBUFFERSIZE, "invalid tcp buffer size.");
		if ((nSendBufferSize < TCPMINBUFFERSIZE) || (nSendBufferSize > TCPMAXBUFFERSIZE))
			throw CException (eErrorCode::INVALIDTCPBUFFERSIZE, "invalid tcp buffer size.");

		m_pImpl.reset ( new CTcpConnectionImpl () );
		m_ReceiveBuffer.resize (nReceiveBufferSize);
		m_SendBuffer1.resize (nSendBufferSize);
		m_SendBuffer2.resize (nSendBufferSize);
		m_pSendBufferInProcess = m_SendBuffer1.data();
		m_pSendBufferNextInQueue = m_SendBuffer2.data();
	}

	CTcpConnection::~CTcpConnection()
	{

	}

	void CTcpConnection::initialize (uint32_t clientIdent)
	{
		m_pImpl->resetFunctionBlocks ();
		m_ClientIdent = clientIdent;
		m_pImpl->initReceive (m_ClientIdent, m_ReceiveBuffer.data (), m_ReceiveBuffer.size ());
		m_RecvState = eTcpConnectionRecv_State::WAITINGFORDATA;
		m_SendState = eTcpConnectionSend_State::WAITINGFORDATA;
		m_LastError = 0;
		m_SendBufferInProcessSize = 0;
		m_SendBufferNextInQueueSize = 0;
	}

	bool CTcpConnection::canSendData (uint32_t nByteCount)
	{
		if (nByteCount > m_SendBufferMemorySize)
			return false;

		if (m_SendBufferNextInQueueSize + nByteCount > m_SendBufferMemorySize)
			return false;

		return true;
	}

	void CTcpConnection::sendData (uint8_t * pBytes, uint32_t nByteCount)
	{
		if ((pBytes == nullptr) || (nByteCount == 0))
			return;

		if (nByteCount > m_SendBufferMemorySize)
			throw CException (eErrorCode::TCPSENDBUFFERSIZEEXCEEDED, "tcp send byte count exceeds buffer size.");

		if (m_SendBufferNextInQueueSize + nByteCount > m_SendBufferMemorySize)
			throw CException (eErrorCode::TCPSENDBUFFERISFULL, "tcp send buffer is full.");

		uint8_t * pSource = pBytes;
		uint8_t * pTarget = &m_pSendBufferNextInQueue[m_SendBufferNextInQueueSize];
		memcpy (pTarget, pSource, nByteCount);
		m_SendBufferNextInQueueSize += nByteCount;
		queueDataCounter++;
		queueDataBytes += nByteCount;

	}

	void CTcpConnection::handleCyclic ()
	{

		queueLength = m_SendBufferNextInQueueSize;
		sendLength = m_SendBufferInProcessSize;
		currentSendBuffer = (uint8_t*) &m_pSendBufferInProcess[0];
		currentQueueBuffer = (uint8_t*) &m_pSendBufferNextInQueue[0];

		switch (m_RecvState) {

			case eTcpConnectionRecv_State::WAITINGFORDATA:

				if (m_pImpl->tcpRecvIsFinished ()) {
					uint32_t bytesReceived = m_pImpl->tcpBytesReceived ();
					m_pImpl->resetReceive();

					if (bytesReceived > 0) {

						bool bHadError = false;
						uint8_t * pData = m_ReceiveBuffer.data();
						uint32_t bytesToHandle = bytesReceived;
						while ((!bHadError) && (bytesToHandle >= sizeof (TcpIncomingMessage))) {

							if (m_pPacketRegistry->handlePacket (pData, sizeof (TcpIncomingMessage), &m_TempResponse)) {

								TcpOutgoingMessageHeader responseHeader;
								m_TempResponse.buildHeader (responseHeader);

								auto & payLoad = m_TempResponse.getPayload();
								uint32_t nPayLoadSize = m_TempResponse.getCurrentSize();

								sendData ((uint8_t*) &responseHeader, sizeof (responseHeader));
								if (nPayLoadSize > 0)
									sendData (&payLoad[0], nPayLoadSize);

								pData += sizeof (TcpIncomingMessage);
								bytesToHandle -= sizeof (TcpIncomingMessage);

							} else {
								bHadError = true;
							}

						}

						if (bHadError ||(bytesToHandle > 0)) {

							m_RecvState = eTcpConnectionRecv_State::ERROR;

						} else {
							m_RecvState = eTcpConnectionRecv_State::RESETCONNECTION;
						}

					} else {

						m_RecvState = eTcpConnectionRecv_State::RESETCONNECTION;

					}

					totalBytesReceived += bytesReceived;

				} else if (m_pImpl->tcpRecvIsBusy ()) {
					m_RecvState = eTcpConnectionRecv_State::WAITINGFORDATA;
				}
				else {
					m_RecvState = eTcpConnectionRecv_State::ERROR;
					m_LastError = m_pImpl->tcpRecvErrorCode ();
				}

				break;

			case eTcpConnectionRecv_State::RESETCONNECTION:
				m_pImpl->initReceive (m_ClientIdent, m_ReceiveBuffer.data (), m_ReceiveBuffer.size ());
				m_RecvState = eTcpConnectionRecv_State::WAITINGFORDATA;

				break;

			case eTcpConnectionRecv_State::INACTIVE:
				break;

			case eTcpConnectionRecv_State::ERROR:
				break;

			default:
				throw CException (eErrorCode::UNKNOWNTCPRECVSTATE, "tcp connection is in unknown recv state.");
		}

		switch (m_SendState)
		{
			case eTcpConnectionSend_State::WAITINGFORDATA:
				if (m_SendBufferNextInQueueSize > 0) {
					m_SendBufferInProcessSize = m_SendBufferNextInQueueSize;
					m_SendBufferNextInQueueSize = 0;

					std::swap (m_pSendBufferInProcess, m_pSendBufferNextInQueue);

					m_pImpl->initSend (m_ClientIdent, m_pSendBufferInProcess, m_SendBufferInProcessSize);

					m_SendState = eTcpConnectionSend_State::SENDING;

				} else {
					m_SendState = eTcpConnectionSend_State::WAITINGFORDATA;
				}
				break;

			case eTcpConnectionSend_State::SENDING:

				if (m_pImpl->tcpSendIsFinished ())
				{
					uint32_t bytesSent = m_pImpl->tcpBytesSent ();
					m_pImpl->resetSend ();
					m_SendState = eTcpConnectionSend_State::WAITINGFORDATA;

				} else if (m_pImpl->tcpSendIsBusy ())
				{
					m_SendState = eTcpConnectionSend_State::SENDING;
				} else {
					m_SendState = eTcpConnectionSend_State::ERROR;
				}

				break;

			case eTcpConnectionSend_State::INACTIVE:
				break;

			case eTcpConnectionSend_State::ERROR:
				break;

			default:
				throw CException (eErrorCode::UNKNOWNTCPSENDSTATE, "tcp connection is in unknown send state.");
		}

		m_pImpl->handleCyclic ();
	}

	CTcpServer::CTcpServer (uint32_t port, uint32_t maxConnections, uint32_t nPacketSignature)
		: m_State (eTcpServer_State::INACTIVE), m_Port (port), m_LastError (0), m_MaxConnections (maxConnections)
	{
		m_pImpl.reset ( new CTcpServerImpl () );
		m_PacketRegistry.reset (new CTcpPacketRegistry (nPacketSignature));

		for (uint32_t nIndex = 0; nIndex < m_MaxConnections; nIndex++) {
			m_InactiveConnections.push_back (std::make_shared<CTcpConnection> (1024, 1024*1024, m_PacketRegistry.get()));
		}

	}

CTcpServer::~CTcpServer()
{

}

bool CTcpServer::serverRunning ()
{
	return (m_State != eTcpServer_State::INACTIVE);
}

bool CTcpServer::clientConnected ()
{
	throw CException (eErrorCode::NOTIMPLEMENTED, "not implemented");
	//return (m_TcpServer.identclnt != 0);
}

void CTcpServer::startServer ()
{
	if (m_State != eTcpServer_State::INACTIVE)
		throw CException (eErrorCode::SERVERISALREADYRUNNING, "server is already running");

	m_State = eTcpServer_State::INIT;
}

void CTcpServer::stopServer ()
{
	if (m_State == eTcpServer_State::INACTIVE)
		throw CException (eErrorCode::SERVERISALREADYRUNNING, "server is already stopped");

	m_State = eTcpServer_State::INACTIVE;
}

bool CTcpServer::enableConnection (uint32_t nClientIdent)
{
	if (m_InactiveConnections.empty ()) {
		return false;
	}

	auto iIter = m_InactiveConnections.begin ();
	auto pConnection = *iIter;
	m_InactiveConnections.erase (iIter);

	pConnection->initialize (nClientIdent);
	m_ActiveConnections.push_back (pConnection);

	return true;

}

void CTcpServer::handleServer ()
{

	switch (m_State) {
		case eTcpServer_State::INIT:
			m_pImpl->initialiseTCP (m_Port);
			m_State = eTcpServer_State::INITIALIZING;
			break;

		case eTcpServer_State::INITIALIZING:

			if (m_pImpl->tcpOpenIsFinished ()) {
				m_pImpl->listenOnSocket (m_pImpl->tcpOpenIdent (), m_MaxConnections);
				m_State = eTcpServer_State::LISTENING;

			} else if (m_pImpl->tcpOpenIsBusy ()) {
				m_State = eTcpServer_State::INITIALIZING;

			}
			else {

				m_State = eTcpServer_State::ERROR;
				m_LastError = m_pImpl->tcpOpenErrorCode ();
			}

			break;

		case eTcpServer_State::LISTENING:

			if (m_pImpl->tcpListenClientConnected ()) {

				uint32_t nClientIdent = m_pImpl->tcpListenClientIdent ();

				if (enableConnection (nClientIdent)) {
					m_State = eTcpServer_State::LISTENING;
				} else {
					//  Too many connections!
					m_pImpl->closeClientConnection (nClientIdent);
					m_State = eTcpServer_State::CLOSINGCONNECTION;
				}

			} else if (m_pImpl->tcpListenIsBusy ()) {
				m_State = eTcpServer_State::LISTENING;

			}
			else {

				m_State = eTcpServer_State::ERROR;
				m_LastError = m_pImpl->tcpListenErrorCode ();
			}

			break;

		case eTcpServer_State::CLOSINGCONNECTION:
				if (m_pImpl->tcpCloseFinished ()) {

					m_pImpl->resetClose ();
					m_State = eTcpServer_State::LISTENING;

				} else if (m_pImpl->tcpCloseIsBusy ()) {
					m_State = eTcpServer_State::CLOSINGCONNECTION;

				}
				else {

					m_State = eTcpServer_State::ERROR;
					m_LastError = m_pImpl->tcpCloseErrorCode ();
				}
			break;

		case eTcpServer_State::INACTIVE:
			break;

		case eTcpServer_State::ERROR:
			break;

		default:
			throw CException (eErrorCode::UNKNOWNTCPSERVERSTATE, "tcp server is in unknown state.");

		};

	for (auto pConnection : m_ActiveConnections)
		pConnection->handleCyclic ();

	m_pImpl->handleCyclic ();

}

void * CTcpServer::getFunctionBlockOpen ()
{
	return m_pImpl->getFunctionBlockOpen ();
}

void * CTcpServer::getFunctionBlockClose ()
{
	return m_pImpl->getFunctionBlockClose ();
}

void * CTcpServer::getFunctionBlockServer ()
{
	return m_pImpl->getFunctionBlockServer ();
}

void CTcpServer::registerPacketHandler (std::shared_ptr<CTcpPacketHandler> pPacketHandler)
{
	m_PacketRegistry->registerHandler (pPacketHandler);
}

CTcpPacketRegistry * CTcpServer::getPacketRegistry ()
{
	return m_PacketRegistry.get ();
}

}
```
